// TwinCAT 3 PLC project tc_project_app
// ProgramVersion: 3.1.4024.12
// libraries:
//   Tc2_EtherCAT, * (Beckhoff Automation GmbH)
//   Tc2_MC2, * (Beckhoff Automation GmbH)
//   Tc2_Standard, * (Beckhoff Automation GmbH)
//   Tc2_SUPS, * (Beckhoff Automation GmbH)
//   Tc2_System, * (Beckhoff Automation GmbH)
//   Tc2_Utilities, * (Beckhoff Automation GmbH)
//   Tc3_MC2_AdvancedHoming, * (Beckhoff Automation GmbH)
//   Tc3_Module, * (Beckhoff Automation GmbH)
//   VisuDialogs, * (System)
// project tree:
//   DUTs/Bridge Terminal PDOs/ ST_Bridge_TSCS_OUTPUTS.TcDUT, ST_Bridge_TSCS_INPUTS.TcDUT
//   DUTs/ E_HOME_STATE.TcDUT, E_MOTION_MODE.TcDUT (not stored), E_OPERATION_MODE.TcDUT (not stored), E_OPERATION_MODE_NO.TcDUT (not stored), E_PHASE_TYPE.TcDUT (not stored), E_PWM_TYPE.TcDUT, E_PHASING_STATE_MACHINE.TcDUT (not stored), E_POSITIONING_STATE_MACHINE.TcDUT (not stored), E_VELOCITY_STATE_MACHINE.TcDUT, ST_INDRADRIVE_AXIS_COMMAND.TcDUT, ST_INDRADRIVE_AXIS_STATUS.TcDUT, ST_HW_CONTROL_ROT.TcDUT, ST_HW_CONTROL_XYZ.TcDUT, ST_HW_STATUS_DEV.TcDUT, ST_HW_STATUS_XYZ.TcDUT, ST_INDRADRIVE_IO_INPUT.TcDUT, ST_INDRADRIVE_IO_OUTPUT.TcDUT (not stored), ST_S134_MASTERCONTROLWORD.TcDUT (not stored), ST_S135_DRIVESTATUSWORD.TcDUT (not stored), ST_S144_SIGNALSTATUSWORD.TcDUT, ST_S145_SIGNALCONTROLWORD.TcDUT, ST_HW_STATUS_ROT.TcDUT, ST_STATUS_ROT.TcDUT, ST_TMS_INTERLOCKS.TcDUT, TARGET_STATE_MACHINE.TcDUT
//   / GlobalTextList.TcGTLO, PlcTask.TcTTO, PlcTaskCom.TcTTO, Visualization Manager.TcVMO (not stored)
//   GVLs/ GVL_Bridge_TSCS.TcGVL, GVL_APP.TcGVL, GVL_ErrorCodes.TcGVL, GVL_Parameters.TcGVL
//   POUs/Application_Specific/Applications/ Application_Template.TcPOU
//   POUs/Application_Specific/Axes/ Axis_Template.TcPOU, Axis_1.TcPOU, Axis_2.TcPOU, Axis_3.TcPOU
//   POUs/Bridge Terminal/FBs/ FB_Bridge_Outputs_Real.TcPOU, FB_Bridge_Inputs_Real.TcPOU, OSCAT_BYTE_OF_BIT.TcPOU, OSCAT_BYTE_TO_BITS.TcPOU, OSCAT_DW_TO_REAL.TcPOU, OSCAT_REAL_TO_DW.TcPOU
//   POUs/Bridge Terminal/ TSCS_Bridge_Inputs.TcPOU, TSCS_Bridge_Outputs.TcPOU, TSCS_Bridge_Diagnostic.TcPOU
//   POUs/Common/ChangeConfig/ FB_ReadFloatParameter.TcPOU, FB_ReadParameterInNc_v1_00.TcPOU, FB_WriteFloatParameter.TcPOU, FB_WriteParameterInNc_v1_00.TcPOU
//   POUs/Common/ErrorHandling/ DUT_ErrorState.TcDUT, FB_ErrorSystem.TcPOU (not stored), FB_GenericError.TcPOU, FB_NC_Error.TcPOU, FB_TerminalError.TcPOU, ST_ErrorEntry.TcDUT, ST_ErrorSystem.TcDUT
//   POUs/Common/GVLs_std/ GVL_back.TcGVL (not stored)
//   POUs/Common/Hardware/EtherCAT_Terminals/Analog_Inputs/ EL3174_0002.TcPOU, EL3214.TcPOU, EL3255.TcPOU, El3742.TcPOU
//   POUs/Common/Hardware/EtherCAT_Terminals/Communication/ EL6695.TcPOU
//   POUs/Common/Hardware/EtherCAT_Terminals/Digital_Inputs/ EL1008.TcPOU, EL1018.TcPOU, EL1252.TcPOU, EL1808.TcPOU, EL1809.TcPOU, EL1819.TcPOU
//   POUs/Common/Hardware/EtherCAT_Terminals/Digital_Outputs/ EL2014.TcPOU, EL2032.TcPOU, EL2252.TcPOU, EL2808.TcPOU, EL2819.TcPOU
//   POUs/Common/Hardware/EtherCAT_Terminals/Digital_Outputs/External_Types/ dutEL2521_Ctrl.TcDUT, dutEL2521_Status.TcDUT
//   POUs/Common/Hardware/EtherCAT_Terminals/Drives/ EL2522.TcPOU, EL4134.TcPOU, EL7037.TcPOU, EL7041_0052.TcPOU, EL7047.TcPOU, EL7211.TcPOU, indraDrive.TcPOU, iPOS8020.TcPOU
//   POUs/Common/Hardware/EtherCAT_Terminals/Feedback_Terminals/ EL5002.TcPOU, EL5021.TcPOU, EL5042.TcPOU, EL5101.TcPOU, EL7201.TcPOU
//   POUs/Common/Hardware/EtherCAT_Terminals/System/ EK1100.TcPOU, EK1110.TcPOU, EL9410.TcPOU, EL9505.TcPOU
//   POUs/Data Type Conversion Functions/ SCALE_REAL_TO_UDINT.TcPOU, SCALE_UDINT_TO_REAL.TcPOU
//   POUs/ MAIN_NORMAL_MOTION.TcPOU, MAIN.TcPOU
//   POUs/Target/ fbIndraDrive.TcPOU, FB_ModePhasing.TcPOU, FB_CalcVeloFromLatch.TcPOU, FB_ModeVelo.TcPOU, FB_ModePos.TcPOU, FB_ModeHome.TcPOU, FB_PID.TcPOU, FB_RampVelo.TcPOU, FB_PWM.TcPOU, FB_TargetSuperImpose.TcPOU (not stored)
//   tc_mca_std_lib_real/DUTs/ E_AxisParameters.TcTLEO (not stored), E_EncoderTypeClass.TcDUT (not stored), E_HomeSwitchTypeClass.TcDUT (not stored), E_HomingRoutines.TcTLEO (not stored), E_MotionFunctions.TcDUT (not stored), E_MotorTypeClass.TcDUT (not stored), E_RestorePosition.TcDUT (not stored), ST_AxisConfig.TcDUT (not stored), ST_AxisControl.TcDUT (not stored), ST_AxisDescription.TcDUT (not stored), ST_AxisError.TcDUT (not stored), ST_AxisInputs.TcDUT (not stored), ST_AxisPersistent.TcDUT (not stored), ST_AxisStatus.TcDUT (not stored), ST_AxisStruct.TcDUT (not stored), ST_GearAxis.TcDUT (not stored)
//   tc_mca_std_lib_real/GVLs/ GVL.TcGVL (not stored)
//   tc_mca_std_lib_real/POUs/Motion/ FB_Axis.TcPOU (not stored)
//   tc_mca_std_lib_real/POUs/Motion/Homing/ FB_Homing.TcPOU (not stored)
//   tc_mca_std_lib_real/VISUs/ languageSupport.TcTLO (not stored), MainVisu.TcVIS (not stored), visuTextLinks.TcTLO (not stored)
//   tc_pils/tc_pils_app_specific/GVLs/ GVL_PILS.TcGVL (not stored)
//   tc_pils/tc_pils_app_specific/POUs/ PILS_DEVICES.TcPOU (not stored)
//   tc_pils/tc_pils_generic/DUTs/ E_Permission.TcDUT (not stored), E_PILS_ParamControl.TcDUT (not stored), E_PILS_State.TcDUT (not stored), ST_1201.TcDUT (not stored), ST_1202.TcDUT (not stored), ST_1204.TcDUT (not stored), ST_1602.TcDUT (not stored), ST_5008.TcDUT (not stored), ST_5010.TcDUT (not stored), ST_AxisParameters.TcDUT (not stored), ST_DeviceInfo.TcDUT (not stored), ST_Indexer.TcDUT (not stored), ST_Indexer_InfoTyp0.TcDUT (not stored), ST_ParamOutput.TcDUT (not stored), U_IndexerData.TcDUT (not stored)
//   tc_pils/tc_pils_generic/POUs/ COMM.TcPOU (not stored)
//   tc_pils/tc_pils_generic/POUs/PILS_device_types/ FB_5008_Axis.TcPOU (not stored), FB_5010_Axis.TcPOU (not stored)
// real-time tasks:
//   TASK PlcTaskCom: cycle T#1ms, priority 26, ADS port 350
//   TASK PlcTask: cycle T#1ms, priority 20, ADS port 351
//   TASK Task faster: cycle T#1ms, priority 1, ADS port 352
// motion (NC):
//   TASK NC-Task 1 SAF: cycle T#2ms, priority 4, ADS port 501
//   TASK NC-Task 1 SVB: cycle T#10ms, priority 8, ADS port 511
//   AXIS Axis 1 (id 1)
//     Dynamic: AccelerationMaximum=0.15, DecelerationMaximum=0.15, Acceleration=0.02, Deceleration=0.02, Jerk=10
//     Velo: RefSearch=0.1, RefSync=0.1, SlowManual=0.01, FastManual=0.05, Maximum=0.3
//     PositionAreaControl: Range=0.2
//     TargetPosControl: Range=0.2
//     OtherSettings: AllowMotionCmdToSlave=true, PulseDistancePos=0.1, PulseDistanceNeg=0.1
//     encoder EncType=19
//       EncPara: ScaleFactorNumerator=0.340251786, ScaleFactorDenominator=51200, Inverse=true, MaxCount=#xffffffff
//     drive DrvType=16
//       DrvPara: Inverse=true, MaxCount=#xffffffff
//         Analog: VeloReferenz=0.3, VeloScale=8192, TorqueSetpointScale=10, ScaleFactorActTorque=0.1
//         TimeComp: TaskDelayCycles=1
//     controller CtrType=1
//       CtrPara: PriorControlFactor=1
//         PosDiffControl: Range=0.2, Time=0.1
//         PID: PosKp=0.1
//         Observer: BandWidth=20
//   AXIS Axis 2 (id 2)
//     Dynamic: AccelerationMaximum=0.15, DecelerationMaximum=0.15, Acceleration=0.02, Deceleration=0.02, Jerk=10
//     Velo: RefSearch=0.1, RefSync=0.1, SlowManual=0.01, FastManual=0.05, Maximum=0.3
//     PositionAreaControl: Range=0.2
//     TargetPosControl: Range=0.2
//     OtherSettings: AllowMotionCmdToSlave=true, PulseDistancePos=0.1, PulseDistanceNeg=0.1
//     encoder EncType=19
//       EncPara: ScaleFactorNumerator=0.340251786, ScaleFactorDenominator=51200, Inverse=true, MaxCount=#xffffffff
//     drive DrvType=16
//       DrvPara: Inverse=true, MaxCount=#xffffffff
//         Analog: VeloReferenz=0.3, VeloScale=8192, TorqueSetpointScale=10, ScaleFactorActTorque=0.1
//         TimeComp: TaskDelayCycles=1
//     controller CtrType=1
//       CtrPara: PriorControlFactor=1
//         PosDiffControl: Range=0.2, Time=0.1
//         PID: PosKp=0.1
//         Observer: BandWidth=20
//   AXIS Axis 3 (id 3)
//     Dynamic: AccelerationMaximum=0.03, DecelerationMaximum=0.03, Acceleration=0.01, Deceleration=0.01, Jerk=10
//     Velo: RefSearch=0.01, RefSync=0.01, SlowManual=0.01, FastManual=0.02, Maximum=0.05
//     PositionAreaControl: Range=0.01
//     TargetPosControl: Range=0.01
//     OtherSettings: AllowMotionCmdToSlave=true, PulseDistancePos=0.02, PulseDistanceNeg=0.02
//     encoder EncType=19
//       EncPara: ScaleFactorNumerator=0.011468, ScaleFactorDenominator=51200, MaxCount=#xffffffff
//     drive DrvType=16
//       DrvPara: MaxCount=#xffffffff
//         Analog: VeloReferenz=0.05, VeloScale=8192, TorqueSetpointScale=10, ScaleFactorActTorque=0.1
//         TimeComp: TaskDelayCycles=1
//     controller CtrType=1
//       CtrPara: PriorControlFactor=1
//         PosDiffControl: Range=0.01, Time=0.1
//         PID: PosKp=0.1
//         Observer: BandWidth=20
// I/O:
//   DEVICE Device 1 (EtherCAT), AmsNetId 172.30.2.35.2.1
//     Term 1 (EK1200) [EK1200-5000 EtherCAT Power supply (2A E-Bus)]
//       Term 2 (EL1809) [EL1809 16Ch. Dig. Input 24V, 3ms]
//       Term 3 (EL1809) [EL1809 16Ch. Dig. Input 24V, 3ms]
//       Term 4 (EL2819) [EL2819 16Ch. Dig. Output 24V, 0,5A, Diagnostic]
//       Term 5 (EL2819) [EL2819 16Ch. Dig. Output 24V, 0,5A, Diagnostic]
//       Term 6 (EL9505) [EL9505 Power supply terminal 5V]
//       Term 7 (EL1252-0050) [EL1252-0050 2Ch. Fast Dig. Input 5V, 1µs, DC Latch]
//       Term 8 (EL9410) [EL9410 E-Bus Power Supplier  (Diagnostics)]
//       Term 9 (EL1252) [EL1252 2Ch. Fast Dig. Input 24V, 1µs, DC Latch]
//       Term 10 (EL7201) [EL7201 1Ch. MDP742 Servo motor output stage (50V, 4A)]
//       Term 11 (EL7201) [EL7201 1Ch. MDP742 Servo motor output stage (50V, 4A)]
//       Term 12 (EL7201) [EL7201 1Ch. MDP742 Servo motor output stage (50V, 4A)]
//       Term 13 (EL3214) [EL3214 4Ch. Ana. Input PT100 (RTD)]
//       Term 18 (EL5021) [EL5021 1Ch. Sin/Cos Encoder]
//       Term 14 (EL6695) [EL6695 EtherCAT Bridge terminal (Primary)]
//       Term 15 (EL9410) [EL9410 E-Bus Power Supplier  (Diagnostics)]
//       Term 16 (EL2032) [EL2032 2Ch. Dig. Output 24V, 2A, Diagnostic]
//       Term 17 (EK1110) [EK1110 EtherCAT extension]
//     Drive 10 (IndraDrive MPB18/19) [IndraDrive MPB18/19]
//     Drive 49 (iPOS8020 BX-CAT) [iPOS8020 BX-CAT]
//     Drive 50 (iPOS8020 BX-CAT) [iPOS8020 BX-CAT]
//     Drive 51 (iPOS8020 BX-CAT) [iPOS8020 BX-CAT]
// variable links:
//   (this object) <-> Device 1 (EtherCAT)/Drive 49 (iPOS8020 BX-CAT)
//     Drive/Inputs/In/nDataIn1 <-> Transmit PDO 2 mapping parameters/Following error actual value
//     Drive/Inputs/In/nDataIn3[0] <-> Transmit PDO 1 mapping parameters/Torque (current) actual value
//     Drive/Inputs/In/nDcOutputTime <-> InfoData/DcOutputShift
//     Drive/Inputs/In/nState1 <-> Transmit PDO 1 mapping parameters/Statusword
//     Drive/Inputs/In/nState2 <-> Transmit PDO 1 mapping parameters/Statusword @bit 8
//     Drive/Inputs/In/nState4 @bit 1 <-> WcState/InputToggle
//     Drive/Inputs/In/nState4 <-> WcState/WcState
//     Drive/Outputs/Out/nCtrl1 <-> Receive PDO 1 mapping parameters/Controlword
//     Drive/Outputs/Out/nCtrl2 <-> Receive PDO 1 mapping parameters/Controlword @bit 8
//     Drive/Outputs/Out/nDataOut2 <-> Receive PDO 1 mapping parameters/Target Velocity
//     Enc/Inputs/In/nDataIn1 <-> Transmit PDO 1 mapping parameters/Position actual value
//     Enc/Inputs/In/nDataIn7 <-> Transmit PDO 3 mapping parameters/Velocity actual value
//     Enc/Inputs/In/nDcInputTime <-> InfoData/DcInputShift
//     Enc/Inputs/In/nState4 @bit 1 <-> WcState/InputToggle
//     Enc/Inputs/In/nState4 <-> WcState/WcState
//   (this object) <-> Device 1 (EtherCAT)/Drive 50 (iPOS8020 BX-CAT)
//     Drive/Inputs/In/nDataIn1 <-> Transmit PDO 2 mapping parameters/Following error actual value
//     Drive/Inputs/In/nDataIn3[0] <-> Transmit PDO 1 mapping parameters/Torque (current) actual value
//     Drive/Inputs/In/nDcOutputTime <-> InfoData/DcOutputShift
//     Drive/Inputs/In/nState1 <-> Transmit PDO 1 mapping parameters/Statusword
//     Drive/Inputs/In/nState2 <-> Transmit PDO 1 mapping parameters/Statusword @bit 8
//     Drive/Inputs/In/nState4 @bit 1 <-> WcState/InputToggle
//     Drive/Inputs/In/nState4 <-> WcState/WcState
//     Drive/Outputs/Out/nCtrl1 <-> Receive PDO 1 mapping parameters/Controlword
//     Drive/Outputs/Out/nCtrl2 <-> Receive PDO 1 mapping parameters/Controlword @bit 8
//     Drive/Outputs/Out/nDataOut2 <-> Receive PDO 1 mapping parameters/Target Velocity
//     Enc/Inputs/In/nDataIn1 <-> Transmit PDO 1 mapping parameters/Position actual value
//     Enc/Inputs/In/nDataIn7 <-> Transmit PDO 3 mapping parameters/Velocity actual value
//     Enc/Inputs/In/nDcInputTime <-> InfoData/DcInputShift
//     Enc/Inputs/In/nState4 @bit 1 <-> WcState/InputToggle
//     Enc/Inputs/In/nState4 <-> WcState/WcState
//   (this object) <-> Device 1 (EtherCAT)/Drive 51 (iPOS8020 BX-CAT)
//     Drive/Inputs/In/nDataIn1 <-> Transmit PDO 2 mapping parameters/Following error actual value
//     Drive/Inputs/In/nDataIn3[0] <-> Transmit PDO 1 mapping parameters/Torque (current) actual value
//     Drive/Inputs/In/nDcOutputTime <-> InfoData/DcOutputShift
//     Drive/Inputs/In/nState1 <-> Transmit PDO 1 mapping parameters/Statusword
//     Drive/Inputs/In/nState2 <-> Transmit PDO 1 mapping parameters/Statusword @bit 8
//     Drive/Inputs/In/nState4 @bit 1 <-> WcState/InputToggle
//     Drive/Inputs/In/nState4 <-> WcState/WcState
//     Drive/Outputs/Out/nCtrl1 <-> Receive PDO 1 mapping parameters/Controlword
//     Drive/Outputs/Out/nCtrl2 <-> Receive PDO 1 mapping parameters/Controlword @bit 8
//     Drive/Outputs/Out/nDataOut2 <-> Receive PDO 1 mapping parameters/Target Velocity
//     Enc/Inputs/In/nDataIn1 <-> Transmit PDO 1 mapping parameters/Position actual value
//     Enc/Inputs/In/nDataIn7 <-> Transmit PDO 3 mapping parameters/Velocity actual value
//     Enc/Inputs/In/nDcInputTime <-> InfoData/DcInputShift
//     Enc/Inputs/In/nState4 @bit 1 <-> WcState/InputToggle
//     Enc/Inputs/In/nState4 <-> WcState/WcState
//   tc_project_app Instance <-> Device 1 (EtherCAT)/Drive 10 (IndraDrive MPB18/19)
//     PlcTask Inputs/MAIN.dLatchedPosition <-> AT/Probe value 1 positive edge
//     PlcTask Inputs/MAIN.fbIndraDrive.stDriveStatus.nP173_MarkerPosition <-> AT/Marker position A
//     PlcTask Inputs/MAIN.fbIndraDrive.stDriveStatus.nS135_DriveStatusWord <-> AT/Drive status word
//     PlcTask Inputs/MAIN.fbIndraDrive.stDriveStatus.nS189_PositionError <-> AT/Following distance
//     PlcTask Inputs/MAIN.fbIndraDrive.stDriveStatus.nS386_ActivePositionFeedbackValue <-> AT/Active position feedback value
//     PlcTask Inputs/MAIN.fbIndraDrive.stDriveStatus.nS390_DiagnosticMessageNumber <-> AT/Diagnostic message number
//     PlcTask Inputs/MAIN.fbIndraDrive.stDriveStatus.nS40_VelocityFeedbackValue <-> AT/Velocity feedback value
//     PlcTask Inputs/MAIN.fbIndraDrive.stDriveStatus.nS51_PositionFeedbackValue <-> AT/Position feedback value 1
//     PlcTask Inputs/MAIN.fbIndraDrive.stDriveStatus.nS84_TorqueFeedback <-> AT/Torque/force feedback value
//     PlcTask Inputs/MAIN.fbIndraDrive.stDriveStatus.stS144_SignalStatusWord <-> AT/Signal status word
//     PlcTask Inputs/MAIN.fb_s19_IndraDrive.InfoData_State <-> InfoData/State
//     PlcTask Inputs/MAIN.fb_s19_IndraDrive.WcState_WcState <-> WcState/WcState
//     PlcTask Outputs/MAIN.fbIndraDrive.stDriveCommands.nS108_FeedrateOverride <-> MDT/Feedrate override
//     PlcTask Outputs/MAIN.fbIndraDrive.stDriveCommands.nS258_TargetPosition <-> MDT/Target position
//     PlcTask Outputs/MAIN.fbIndraDrive.stDriveCommands.nS259_PositioningVelocity <-> MDT/Positioning velocity
//     PlcTask Outputs/MAIN.fbIndraDrive.stDriveCommands.nS260_PositioningAcceleration <-> MDT/Ramp 1 pitch
//     PlcTask Outputs/MAIN.fbIndraDrive.stDriveCommands.nS282_PositioningCommandValue <-> MDT/Positioning command value
//     PlcTask Outputs/MAIN.fbIndraDrive.stDriveCommands.nS359_PositioningDeceleration <-> MDT/Deceleration ramp 1
//     PlcTask Outputs/MAIN.fbIndraDrive.stDriveCommands.nS40_VelocityCommandValue <-> MDT/Velocity command value
//     PlcTask Outputs/MAIN.fbIndraDrive.stDriveCommands.nS47_PositionCommandValue <-> MDT/Position command value
//     PlcTask Outputs/MAIN.fbIndraDrive.stDriveCommands.nS92_BiPolarTorqueLimit <-> MDT/Bipolar torque/force limit value
//     PlcTask Outputs/MAIN.fbIndraDrive.stDriveCommands.stS134_MasterControlWord <-> MDT/Master control word
//     PlcTask Outputs/MAIN.fbIndraDrive.stDriveCommands.stS145_SignalControlWord <-> MDT/Signal control word
//     PlcTask Outputs/MAIN.nAdditiveTorqueSetpoint <-> MDT/Additive torque/force command value
//     PlcTaskCom Outputs/MAIN.iTorqueCommandValue <-> MDT/Torque/force command value
//   tc_project_app Instance <-> Device 1 (EtherCAT)/Drive 49 (iPOS8020 BX-CAT)
//     PlcTask Inputs/MAIN.fb_s20_IPOS8020.InfoData_State <-> InfoData/State
//   tc_project_app Instance <-> Device 1 (EtherCAT)/Drive 50 (iPOS8020 BX-CAT)
//     PlcTask Inputs/MAIN.fb_s21_IPOS8020.InfoData_State <-> InfoData/State
//   tc_project_app Instance <-> Device 1 (EtherCAT)/Drive 51 (iPOS8020 BX-CAT)
//     PlcTask Inputs/MAIN.fb_s22_IPOS8020.InfoData_State <-> InfoData/State
//   tc_project_app Instance <-> Device 1 (EtherCAT)/Term 1 (EK1200)/Term 10 (EL7201)
//     PlcTask Inputs/MAIN.fb_s10_EL7201.InfoData_State <-> InfoData/State
//     PlcTask Inputs/MAIN.fb_s10_EL7201.WcState_WcState <-> WcState/WcState
//     PlcTask Inputs/MAIN.fb_s10_EL7201.fPosAct <-> FB Position/Position
//   tc_project_app Instance <-> Device 1 (EtherCAT)/Term 1 (EK1200)/Term 11 (EL7201)
//     PlcTask Inputs/MAIN.fb_s11_EL7201.InfoData_State <-> InfoData/State
//     PlcTask Inputs/MAIN.fb_s11_EL7201.WcState_WcState <-> WcState/WcState
//     PlcTask Inputs/MAIN.fb_s11_EL7201.fPosAct <-> FB Position/Position
//   tc_project_app Instance <-> Device 1 (EtherCAT)/Term 1 (EK1200)/Term 12 (EL7201)
//     PlcTask Inputs/MAIN.fb_s12_EL7201.InfoData_State <-> InfoData/State
//     PlcTask Inputs/MAIN.fb_s12_EL7201.WcState_WcState <-> WcState/WcState
//     PlcTask Inputs/MAIN.fb_s12_EL7201.fPosAct <-> FB Position/Position
//   tc_project_app Instance <-> Device 1 (EtherCAT)/Term 1 (EK1200)/Term 13 (EL3214)
//     PlcTask Inputs/MAIN.fb_s13_EL3214.InfoData_State <-> InfoData/State
//     PlcTask Inputs/MAIN.fb_s13_EL3214.WcState_WcState <-> WcState/WcState
//     PlcTask Inputs/MAIN.fb_s13_EL3214.iAI_{1..4} <-> RTD Inputs Channel {1..4}/Value  (4 links)
//     PlcTask Inputs/MAIN.fb_s13_EL3214.wCh{1..4}_Status <-> RTD Inputs Channel {1..4}/Status  (4 links)
//   tc_project_app Instance <-> Device 1 (EtherCAT)/Term 1 (EK1200)/Term 14 (EL6695)
//     PlcTask Inputs/GVL_Bridge_TSCS.INPUTS/TDU_TestSignal_RB <-> IO Inputs/TDU_WatchDog_RB
//     PlcTask Inputs/GVL_Bridge_TSCS.INPUTS/TSCS_Byte <-> IO Inputs/TSCS_Byte
//     PlcTask Inputs/GVL_Bridge_TSCS.INPUTS/TSCS_Real <-> IO Inputs/TSCS_Real
//     PlcTask Inputs/MAIN.fb_s15_EL6695.InfoData_State <-> InfoData/State
//     PlcTask Inputs/MAIN.fb_s15_EL6695.WcState_WcState <-> WcState/WcState
//     PlcTask Outputs/GVL_Bridge_TSCS.OUTPUTS/TDU_Byte <-> IO Outputs/TDU_Byte
//     PlcTask Outputs/GVL_Bridge_TSCS.OUTPUTS/TDU_Real <-> IO Outputs/TDU_Real
//     PlcTask Outputs/GVL_Bridge_TSCS.OUTPUTS/TDU_TestSignal <-> IO Outputs/TDU_WatchDog
//   tc_project_app Instance <-> Device 1 (EtherCAT)/Term 1 (EK1200)/Term 15 (EL9410)
//     PlcTask Inputs/MAIN.fb_s16_EL9410.InfoData_State <-> InfoData/State
//     PlcTask Inputs/MAIN.fb_s16_EL9410.WcState_WcState <-> WcState/WcState
//     PlcTask Inputs/MAIN.fb_s16_EL9410.bUp_Undervoltage <-> Status Up/Undervoltage
//     PlcTask Inputs/MAIN.fb_s16_EL9410.bUs_Undervoltage <-> Status Us/Undervoltage
//   tc_project_app Instance <-> Device 1 (EtherCAT)/Term 1 (EK1200)/Term 16 (EL2032)
//     PlcTask Inputs/MAIN.fb_s17_EL2032.InfoData_State <-> InfoData/State
//     PlcTask Inputs/MAIN.fb_s17_EL2032.WcState_WcState <-> WcState/WcState
//   tc_project_app Instance <-> Device 1 (EtherCAT)/Term 1 (EK1200)/Term 18 (EL5021)
//     PlcTask Inputs/MAIN.fb_s14_EL5021.InfoData_State <-> InfoData/State
//     PlcTask Inputs/MAIN.fb_s14_EL5021.WcState_WcState <-> WcState/WcState
//     PlcTaskCom Inputs/MAIN.nSecondRotEncoder <-> ENC Status/Counter value
//   tc_project_app Instance <-> Device 1 (EtherCAT)/Term 1 (EK1200)/Term 2 (EL1809)
//     PlcTask Inputs/MAIN.fb_s2_EL1809.InfoData_State <-> InfoData/State
//     PlcTask Inputs/MAIN.fb_s2_EL1809.WcState_WcState <-> WcState/WcState
//     PlcTask Inputs/MAIN.fb_s2_EL1809.bBI_{1..16} <-> Channel {1..16}/Input  (16 links)
//   tc_project_app Instance <-> Device 1 (EtherCAT)/Term 1 (EK1200)/Term 3 (EL1809)
//     PlcTask Inputs/MAIN.fb_s3_EL1809.InfoData_State <-> InfoData/State
//     PlcTask Inputs/MAIN.fb_s3_EL1809.WcState_WcState <-> WcState/WcState
//     PlcTask Inputs/MAIN.fb_s3_EL1809.bBI_{1..16} <-> Channel {1..16}/Input  (16 links)
//   tc_project_app Instance <-> Device 1 (EtherCAT)/Term 1 (EK1200)/Term 4 (EL2819)
//     PlcTask Inputs/MAIN.fb_s4_EL2819.InfoData_State <-> InfoData/State
//     PlcTask Inputs/MAIN.fb_s4_EL2819.WcState_WcState <-> WcState/WcState
//     PlcTask Inputs/MAIN.fb_s4_EL2819.bDev_CommonFault <-> DIG Inputs Device/Common Fault
//     PlcTask Inputs/MAIN.fb_s4_EL2819.bDev_MissingVoltage <-> DIG Inputs Device/Missing Voltage
//     PlcTask Inputs/MAIN.fb_s4_EL2819.bDev_Overtemperature <-> DIG Inputs Device/Overtemperature Device
//     PlcTask Inputs/MAIN.fb_s4_EL2819.bDev_UnderVoltage <-> DIG Inputs Device/Undervoltage
//     PlcTask Inputs/MAIN.fb_s4_EL2819.wCH{1..16}_Diag <-> DIG Diag Inputs/Channel {1..16}  (16 links)
//     PlcTask Outputs/MAIN.stHWControlRot.bRotOmronSensor1Feed <-> DIG Outputs/Channel 1/Output
//     PlcTask Outputs/MAIN.stHWControlRot.bRotOmronSensor2Feed <-> DIG Outputs/Channel 2/Output
//   tc_project_app Instance <-> Device 1 (EtherCAT)/Term 1 (EK1200)/Term 5 (EL2819)
//     PlcTask Inputs/MAIN.fb_s5_EL2819.InfoData_State <-> InfoData/State
//     PlcTask Inputs/MAIN.fb_s5_EL2819.WcState_WcState <-> WcState/WcState
//     PlcTask Inputs/MAIN.fb_s5_EL2819.bDev_CommonFault <-> DIG Inputs Device/Common Fault
//     PlcTask Inputs/MAIN.fb_s5_EL2819.bDev_MissingVoltage <-> DIG Inputs Device/Missing Voltage
//     PlcTask Inputs/MAIN.fb_s5_EL2819.bDev_Overtemperature <-> DIG Inputs Device/Overtemperature Device
//     PlcTask Inputs/MAIN.fb_s5_EL2819.bDev_UnderVoltage <-> DIG Inputs Device/Undervoltage
//     PlcTask Inputs/MAIN.fb_s5_EL2819.wCH{1..16}_Diag <-> DIG Diag Inputs/Channel {1..16}  (16 links)
//     PlcTask Outputs/MAIN.stHWControlX.bBrakeReleaseCmd <-> DIG Outputs/Channel 2/Output
//     PlcTask Outputs/MAIN.stHWControlX.bMinMaxFeed <-> DIG Outputs/Channel 1/Output
//     PlcTask Outputs/MAIN.stHWControlX.bMinMinMaxMaxFeed <-> DIG Outputs/Channel 3/Output
//     PlcTask Outputs/MAIN.stHWControlY.bBrakeReleaseCmd <-> DIG Outputs/Channel 6/Output
//     PlcTask Outputs/MAIN.stHWControlY.bMinMaxFeed <-> DIG Outputs/Channel 5/Output
//     PlcTask Outputs/MAIN.stHWControlY.bMinMinMaxMaxFeed <-> DIG Outputs/Channel 7/Output
//     PlcTask Outputs/MAIN.stHWControlZ.bMinMaxFeed <-> DIG Outputs/Channel 9/Output
//     PlcTask Outputs/MAIN.stHWControlZ.bMinMinMaxMaxFeed <-> DIG Outputs/Channel 10/Output
//   tc_project_app Instance <-> Device 1 (EtherCAT)/Term 1 (EK1200)/Term 6 (EL9505)
//     PlcTask Inputs/MAIN.fb_s6_EL9505.InfoData_State <-> InfoData/State
//     PlcTask Inputs/MAIN.fb_s6_EL9505.WcState_WcState <-> WcState/WcState
//     PlcTask Inputs/MAIN.fb_s6_EL9505.bUoPwr_OK <-> Status Uo/Power OK
//     PlcTask Inputs/MAIN.fb_s6_EL9505.bUo_Overload <-> Status Uo/Overload
//   tc_project_app Instance <-> Device 1 (EtherCAT)/Term 1 (EK1200)/Term 7 (EL1252-0050)
//     PlcTask Inputs/MAIN.fb_s7_EL1252.InfoData_State <-> InfoData/State
//     PlcTask Inputs/MAIN.fb_s7_EL1252.WcState_WcState <-> WcState/WcState
//     PlcTask Inputs/MAIN.fb_s7_EL1252.bBI_1 <-> Channel 1/Input
//     PlcTask Inputs/MAIN.fb_s7_EL1252.bBI_2 <-> Channel 2/Input
//   tc_project_app Instance <-> Device 1 (EtherCAT)/Term 1 (EK1200)/Term 8 (EL9410)
//     PlcTask Inputs/MAIN.fb_s8_EL9410.InfoData_State <-> InfoData/State
//     PlcTask Inputs/MAIN.fb_s8_EL9410.WcState_WcState <-> WcState/WcState
//     PlcTask Inputs/MAIN.fb_s8_EL9410.bUp_Undervoltage <-> Status Up/Undervoltage
//     PlcTask Inputs/MAIN.fb_s8_EL9410.bUs_Undervoltage <-> Status Us/Undervoltage
//   tc_project_app Instance <-> Device 1 (EtherCAT)/Term 1 (EK1200)/Term 9 (EL1252)
//     PlcTask Inputs/MAIN.fb_s9_EL1252.InfoData_State <-> InfoData/State
//     PlcTask Inputs/MAIN.fb_s9_EL1252.WcState_WcState <-> WcState/WcState
//     PlcTask Inputs/MAIN.fb_s9_EL1252.bBI_1 <-> Channel 1/Input
//     PlcTask Inputs/MAIN.fb_s9_EL1252.bBI_2 <-> Channel 2/Input
//   tc_project_app Instance <-> NC-Task 1 SAF/Axes/Axis 1
//     PlcTask Inputs/GVL.astAxes[1].Axis.NcToPlc <-> Outputs/ToPlc
//     PlcTask Outputs/GVL.astAxes[1].Axis.PlcToNc <-> Inputs/FromPlc
//   tc_project_app Instance <-> NC-Task 1 SAF/Axes/Axis 2
//     PlcTask Inputs/GVL.astAxes[2].Axis.NcToPlc <-> Outputs/ToPlc
//     PlcTask Outputs/GVL.astAxes[2].Axis.PlcToNc <-> Inputs/FromPlc
//   tc_project_app Instance <-> NC-Task 1 SAF/Axes/Axis 3
//     PlcTask Inputs/GVL.astAxes[3].Axis.NcToPlc <-> Outputs/ToPlc
//     PlcTask Outputs/GVL.astAxes[3].Axis.PlcToNc <-> Inputs/FromPlc

CONFIGURATION tc_project_app
    RESOURCE PLC ON TwinCAT3
        TASK PlcTask(INTERVAL := T#1ms, PRIORITY := 20);
        TASK PlcTaskCom(INTERVAL := T#1ms, PRIORITY := 26);
        PROGRAM MAIN WITH PlcTask : MAIN;
        PROGRAM MAIN_NORMAL_MOTION WITH PlcTask : MAIN_NORMAL_MOTION;
        PROGRAM COMM WITH PlcTaskCom : COMM;
    END_RESOURCE
END_CONFIGURATION

// ---- DUTs/Bridge Terminal PDOs/ST_Bridge_TSCS_OUTPUTS.TcDUT
TYPE ST_Bridge_TSCS_OUTPUTS :
	// 	Outputs from TDU PLC to bridge terminal (to TSCS PLC)
STRUCT
	TDU_TestSignal : UDINT;	// Diagnostic signal (for readback: This PLC -> Other PLC -> This PLC)
	TDU_Byte : ARRAY [0..3] OF BYTE; // Boolean words from TDU PLC (5x 8 Booleans)
	TDU_Real : ARRAY [0..7] OF UDINT;
END_STRUCT
END_TYPE

// ---- DUTs/Bridge Terminal PDOs/ST_Bridge_TSCS_INPUTS.TcDUT
TYPE ST_Bridge_TSCS_INPUTS :
// 	Inputs from bridge terminal (bridge with TSCS PLC)
STRUCT
	TDU_TestSignal_RB : UDINT;				// Diagnostic signal readback TDU->TSCS->TDU
	TSCS_Byte : ARRAY [0..3] OF BYTE;		// Boolean words from TSCS PLC (5x 8 Booleans)
	TSCS_Real : ARRAY [0..7] OF UDINT;
END_STRUCT
END_TYPE

// ---- DUTs/E_HOME_STATE.TcDUT
{attribute 'qualified_only'}
{attribute 'strict'}
TYPE E_HOME_STATE :
(
	IDLE      := 0,
	RAMP_UP   := 1,
	HOMING    := 2,
	RAMP_DOWN := 3
);
END_TYPE

// ---- DUTs/E_PWM_TYPE.TcDUT
{attribute 'qualified_only'}
{attribute 'strict'}
TYPE E_PWM_TYPE :
(
	NONE := 0,
	OPTIMIZED:=1,
	SIMPLE:=2
);
END_TYPE

// ---- DUTs/E_VELOCITY_STATE_MACHINE.TcDUT
{attribute 'qualified_only'}
{attribute 'strict'}
TYPE E_VELOCITY_STATE_MACHINE :
(
	POWER_OFF := 0,
	POWER_ON := 1,
	VELOCITY := 2 
);
END_TYPE

// ---- DUTs/ST_INDRADRIVE_AXIS_COMMAND.TcDUT
TYPE ST_INDRADRIVE_AXIS_COMMAND :
STRUCT
	eOperationMode				: E_OPERATION_MODE_NO	:= E_OPERATION_MODE_NO.ePrimaryOpMode;	// (S134.0-2) Defines the Operation mode to use (the different operation modes are configured in the drive) 
	bEnableAxis					: BOOL	:= FALSE; 	// FALSE (S134.13-15): Disable drive 
													// TRUE (S134.13-15): Enable drive (torque on the motor) 
	bHaltAxis					: BOOL	:= FALSE;	// FALSE (S134.13-15): Drive performs a HALT operation (Deceleration of drive while maintaining the max. acceleration (S-0-0138). Requires bEnableAxis to be TRUE) 
													// TRUE (S134.13-15): Drive is not halted
	eMotionMode					: E_MOTION_MODE		:= E_MOTION_MODE.eStop;	// Defines the type of motion that shall be performed. This is not functional in Operation Mode Drive internal interpolation! 
	//bPositioningMode			: BOOL;				// (S346.2&1 FALSE&FALSE): Activates positioning mode according to current Operation mode 
	//bJogPositive				: BOOL;				// (S346.2&1 FALSE&TRUE): Activates jogging in positive direction  
	//bJogNeagtive				: BOOL;				// (S346.2&1 TRUE&FALSE): Activates jogging in negative direction
	//bStopAxis					: BOOL;				// (S346.2&1 TRUE&TRUE): Stops the axis 
	bCommandPositionChange		: BOOL	:= FALSE;	// (S346.5) FALSE: Drive moves to current target position, before positioning to new target position (when bCommandValueAccept is toggled) 
													// (S346.5) TRUE: Immediate of target position, i.e., drive immediately acknowledges the new target position (when bCommandValueAccept is toggled) 
	fCommandPosition			: LREAL	:= 0.0;		// (S47, S258 or S282 according to OperationMode)
	fCommandVelocity			: LREAL	:= 0.0; 	// (S259): The velocity used for Positioning and Jogging
	fCommandAcceleration		: LREAL	:= 0.0;		// (S260): The acceleration used for Positioning and Jogging 
	fCommandDeceleration		: LREAL	:= 0.0;		// (S359): The deceleration used for Positioning and Jogging 
	fFeedrateOverride			: LREAL	:= 100.0; 	// (S108):  Parameter used for variable adjustment of the velocity [0..100%] 
	fTorqueLimit				: LREAL	:= 100.0;	// (S92):  Parameter used for limiting the torque [0..drive/motor limit%] 
	bPositionCommandValue		: BOOL	:= FALSE;	// (S346.3): FALSE: Command position is absolute 
													// (S346.3): TRUE: Command position is relative
	bCommandValueAccept			: BOOL	:= FALSE; 	// (S346.0) Toggle bit (FALSE->TRUE or TRUE->FALSE) to start a positioning command in Operation mode "Drive controlled Positioning"
	bCmd_ErrorReset				: BOOL	:= FALSE;	// (S99): Reset the error of the drive 
	bCmd_SetAbsolutePosition	: BOOL	:= FALSE;	// (P12, C0300): Sets the Absolute position of the drive according to drive configuration 
	bCmd_DriveControlledHoming	: BOOL	:= FALSE;	// (S148, C0600): Starts the homing procedure configured in the drive. NOTE that this does not set the absolute position 
	bCmd_DisableLimits			: BOOL	:= FALSE;	// (bS159, C1300): Disables Monitoring of Position error, Position command error, Velocity error and Acceleration limit
	bCmd_ActivateParameterMode	: BOOL	:= FALSE;	// (S420, C0400): TRUE: Brings the drive to parameter mode 
	bCmd_ExitParameterMode		: BOOL	:= FALSE;	// (S422, C0200): TRUE: Brings the drive from parameter mode 
	bCmd_RunVirtualMater		: BOOL	:= FALSE;	// Jog command to the virtual Master
	bCmd_NCHomeEnable           : BOOL  := FALSE;   // Home from master NC enable (to be able to latch ref marks)
    bCmd_GetMarkerPosition      : BOOL  := FALSE;   // Start command C1400 Get Marker Position
	fVelocityCommandValue		: LREAL	:= 0.0; 	// (S40): The velocity used for Positioning and Jogging
END_STRUCT
END_TYPE

// ---- DUTs/ST_INDRADRIVE_AXIS_STATUS.TcDUT
TYPE ST_INDRADRIVE_AXIS_STATUS :
STRUCT

	bDriveInParameterMode		: BOOL;		// FALSE (S424): Drive is in Operating mode
											// TRUE (S424): The drive is in parameter mode (parameterization level 1 is active)
	eActualOperationModeNo		: E_OPERATION_MODE_NO	:= E_OPERATION_MODE_NO.ePrimaryOpMode;	// (S134.0-2) Defines the Operation mode to use (the different operation modes are configured in the drive) 
	bDCBusPresent				: BOOL;		// FALSE: DC-bus is not present (drive status bb)
											// TRUE (S135.1&0 TRUE&FALSE): DC-bus present (drive state Ab)
	bAxisEnabled				: BOOL; 	// TRUE (S135.1&0 TRUE&TRUE): Axis is operational with torque (drive state AF)
	bAxisHomedStatus			: BOOL; 	// TRUE (S403.0): Axis absolute position is established 
	bAxisStandStillStatus		: BOOL;		// TRUE (S331): Axis is standing still (velocity below configured threshold) 
	bAxisInTargetPosition		: BOOL;		// TRUE (S437.2): Axis command position is reached
	bAxisConstantVelocityStatus	: BOOL;		// TRUE (S437.4): Axis in constant velocity
	bAxisAccelerationStatus		: BOOL;		// TRUE (S437.5): Axis in acceleration
	bAxisDecelerationStatus		: BOOL;		// TRUE (S437.6): Axis in deceleration
	bAxisJogStatus				: BOOL;		// TRUE (S437.12): Axis in jog mode
	fActualPosition				: LREAL;	// The actual position of the axis
	fActualVelocity				: LREAL;	// The actual velocity of the axis
	fActualTorque				: LREAL;	// The actual torque of the axis
	fPositionError				: LREAL;	// The position error of the axis, i.e. the deviation between the Axis Set position and Actual position
	fMarkerPosition             : LREAL;
    bCommandChange				: BOOL;		// (S135.5): Bit that toggle every time a new command has been recognised by the drive 
	bCommandValueProcessing		: BOOL;		// FALSE (S115.3): Drive ignores (external) command value input (S47, S258, S282 etc) 
											// TRUE (S115.3): Drive follows (external) command value input (S47, S258, S282 etc) 
	bSTOActiveCh1   			: BOOL;     // FALSE: STO OK (motor can run)
	                                        // TRUE:  STO is active
	bSTOActiveCh2   			: BOOL;     // FALSE: STO OK (motor can run)
	                                        // TRUE:  STO is active
    bLimitsDisabled				: BOOL;		// TRUE (S159-C1300): 	Monitoring of Position error, Position command error, Velocity error and Acceleration limit is disabled
											// FALSE (S159-C1300): 	Monitoring of Position error, Position command error, Velocity error and Acceleration limit is enabled 
	bDiagMessage				: BOOL;		// TRUE (S135.11): There is a Diagnostic message on the drive 
	bWarning					: BOOL;		// TRUE (S135.12): There is a warning present on the drive 
	bError 						: BOOL;		// TRUE (S135.13): There is an error present on the drive 
	bCmd_GetMarkerPositionDone  : BOOL;     // C1400 command Get Marker Position done
	nDiagMessage				: DWORD;	// (S390) Displays the actual diagnostic message on the drive 
END_STRUCT
END_TYPE

// ---- DUTs/ST_HW_CONTROL_ROT.TcDUT

TYPE ST_HW_CONTROL_ROT :
STRUCT
	bRotOmronSensor1Feed AT %Q* :BOOL;  // s4: ch1: Feed omron sensor 1
	bRotOmronSensor2Feed AT %Q* :BOOL;  // s4: ch2: Feed omron sensor 2
	bManualInterlockOverride: BOOL:=FALSE;
	bExecute          : BOOL:=FALSE;
	bEnable           : BOOL:=FALSE;
	bReset            : BOOL:=FALSE;
	fVelSet           : LREAL:=0;
	fPosSet           : LREAL:=0;
	eTargetStateCmd   : TARGET_STATE_MACHINE:=TARGET_STATE_MACHINE.NONE;
	ePhaseCntrlAlg    : E_PHASE_TYPE:=E_PHASE_TYPE.PID;
	ePhasePwmType     : E_PWM_TYPE:=E_PWM_TYPE.NONE;
	fPhaseOffsetMM    : LREAL:=0;
	bAllowMotionGUI   : BOOL:=FALSE;       // Allow motion from GUI
	//brake: Only in test rig
	//bBrakeLockOnCmd   : BOOL:=FALSE;
	//bFreeWheelOnOnCmd : BOOL:=TRUE;
	//fBrakeSpNm        : LREAL:=0;
END_STRUCT
END_TYPE

// ---- DUTs/ST_HW_CONTROL_XYZ.TcDUT

TYPE ST_HW_CONTROL_XYZ :
STRUCT
	bMinMaxFeed  AT %Q* :BOOL;         // s5: ch1: kf05: w02.bg01 w02.bg02 stepper x limit switch max, limit min
	bBrakeReleaseCmd  AT %Q* :BOOL;    // s5: ch2: kf05: w02.ql1: stepper x brake ONLY x and Y
	bMinMinMaxMaxFeed  AT %Q* :BOOL;   // s5: ch3: kf05: w02.bg03 w02.bg04 stepper x limit switch max max, limit min min
    bManualInterlockOverride: BOOL:=FALSE;
	bAllowMotionGUI:BOOL:=FALSE;       // Allow motion from GUI
	bExecuteAbsPos:BOOL:=FALSE;
	bExecuteConstVelo:BOOL:=FALSE;
	bExecuteHome:BOOL:=FALSE;
	bExecuteStop:BOOL:=FALSE;
	bEnable:BOOL:=FALSE;
	bExecuteReset:BOOL:=FALSE;
	bJogDirFwd:BOOL:=1;   // 1=fwd, 0=bwd
END_STRUCT
END_TYPE

// ---- DUTs/ST_HW_STATUS_DEV.TcDUT
// HW status for control cabinet alarms and rotation drive
TYPE ST_HW_STATUS_DEV :
STRUCT	
	bEStopOK:BOOL;                       // s2: ch1: emergency stop ok                 Verify: OK   
	bRF02_MainDriveThermalFilterOK:BOOL; // s2: ch2: rf01 termal braking filter OK..   Verify: Q to Markus: Maybe this should be rf02?
	bTA01_TA02_24VSupplyOK:BOOL;         // s2: ch3: ta01 and ta02 24V power supply OK Verify: OK  
	bFC11_Fuse24VOK:BOOL;                // s2: ch4: fc11 24V fuse OK                   Verify: OK
	bFA01_FA02_OvervoltageOK:BOOL;       // s2: ch5: fa01 and fa02 overvoltage protection OK
	bFC01_FuseMainRotationOK:BOOL;       // s2: ch6: fc01 fuse target wheel motor OK
	bFC06_FC07_FuseICSOutletsOK:BOOL;    // s2: ch7: fc06 and fc07 ICS outlets fuse OK
	bFC51_FC52_FC53_FuseUPSOK:BOOL;      // s2: ch8: fc51, fc52 and fc53 UPS fuses OK (something wrong)
	
	// Bridge terminal EL6695
	bBeamOff:BOOL; 
	
END_STRUCT
END_TYPE

// ---- DUTs/ST_HW_STATUS_XYZ.TcDUT
// HW status for XYZ axis
TYPE ST_HW_STATUS_XYZ :
STRUCT
	bEStopOK:BOOL;
	fStepperTemp: LREAL;
	bLimitMax:BOOL;
	bLimitMin:BOOL;
	bLimitMaxMax:BOOL;
	bLimitMinMin:BOOL;
	bSumBwdILOK:BOOL:=FALSE;   
	bSumFwdILOK:BOOL:=FALSE;  
	bManualInterlockOverride:BOOL;
	bHwStatusOK:BOOL;  // Status of hardware (IPOS, EL7201, EL3214, fuses..)
	bGeneralILOK:BOOL:=FALSE;  // All on direction related summary interlocks
	bGeneralAndOverrideILOK:BOOL:=FALSE;
	bBusy:BOOL:=FALSE;
	bEnabled:BOOL:=FALSE;
	bHomed:BOOL:=FALSE;
	bHomingCmdActive:BOOL:=FALSE;
	
	// Position Outside range alarms
	bHiAlm:BOOL:=FALSE;
	bHiHiAlm:BOOL:=FALSE;
	bLoAlm:BOOL:=FALSE;
	bLoLoAlm:BOOL:=FALSE;
	
	//Only X and Y
	bBrakeReleased: BOOL;
	
	//Only for Z
    bLimitMinPark:BOOL;
	bLimitMinMinPark:BOOL;	
	bParkingRangeEnabled:BOOL;
END_STRUCT
END_TYPE

// ---- DUTs/ST_INDRADRIVE_IO_INPUT.TcDUT
TYPE ST_INDRADRIVE_IO_INPUT :	// Contains the data that is read from the drive
STRUCT
	nS135_DriveStatusWord				AT %I*	: ST_S135_DRIVESTATUSWORD; 
	nS51_PositionFeedbackValue			AT %I*	: DINT; 
	nS386_ActivePositionFeedbackValue	AT %I*	: DINT; 
	nS40_VelocityFeedbackValue			AT %I*	: DINT; 
	nS390_DiagnosticMessageNumber		AT %I*	: DWORD; 
	stS144_SignalStatusWord				AT %I*	: ST_S144_SIGNALSTATUSWORD;
	nS84_TorqueFeedback					AT %I*	: INT;
	nS189_PositionError					AT %I*	: DINT;
	nP173_MarkerPosition                AT %I*  : DINT;
END_STRUCT
END_TYPE

// ---- DUTs/ST_S144_SIGNALSTATUSWORD.TcDUT
TYPE ST_S144_SIGNALSTATUSWORD :
STRUCT
	bS424_DriveMode						: BIT; 	// FALSE: Operating mode
												// TRUE: Parameter mode
	{attribute 'hide'}
	bS144_1_NotDefined					: BIT;
	bS403_0_AxisHomedStatus				: BIT; 	// FALSE: Axis is NOT homed 
												// TRUE: Axis is homed
	bS331_StandStillStatus				: BIT; 	// FALSE: Axis is moving
												// TRUE: Axis is standing still 
	bS437_2_CommandPositionReached		: BIT; 	// FALSE: Axis is NOT not within command position
												// TRUE: Axis has reached command position
	{attribute 'hide'}
	bS144_5_NotDefined					: BIT;
	{attribute 'hide'}
	bS144_6_NotDefined					: BIT;
	bP115_3_StatusOfCmdValueProcessing	: BIT; 	// FALSE: Drive ignores external command value input 
												// TRUE: Drive follows external command value input
	
	bP106_1_STO_ch1 					: BIT;  // FALSE: STO OK (motor can run)
	                                            // TRUE:  STO is active
	bP106_2_STO_ch2 					: BIT;  // FALSE: STO OK (motor can run)
	                                            // TRUE:  STO is active
	bS419_0_PositioningCmdAck			: BIT; 	// Toggled as soon as the new Position Command value is accepted and effective
	bS437_4_ConstantVelocity			: BIT; 	// TRUE: Axis in constant velocity
	bS437_5_Acceleration				: BIT; 	// TRUE: Axis in acceleration
	bS437_6_Deceleration				: BIT; 	// TRUE: Axis in deceleration
	bS437_12_JogMode					: BIT; 	// TRUE: Axis in Axis in jog mode
	//{attribute 'hide'}
	//bS144_15_NotDefined					: BIT;	
	bP14_0_C1400_GetMarkerPositionDone  : BIT   := FALSE;
END_STRUCT
END_TYPE

// ---- DUTs/ST_S145_SIGNALCONTROLWORD.TcDUT
TYPE ST_S145_SIGNALCONTROLWORD :
STRUCT
	bS346_0_PosCtrlWord_CmdValueAccept		: BIT	:= FALSE; 	// Toggle to execute Slave Axis command
	bP12_C300_SetAbsolutePosition			: BIT	:= FALSE;	// Sets the Absolute position (defined in S52) of the drive
	bS148_C600_DriveControlledHoming		: BIT	:= FALSE; 	// Initiates the homing procedure defined in the drive
	bS346_3_PosCtrlWord_Abs_Rel				: BIT	:= FALSE;	// FALSE: Absolute 
																// TRUE: Relative									
	bS346_5_PosCtrlWord_ImmBlockChange		: BIT	:= FALSE;	// FALSE: Drive moves to current target position, before positioning at new target position
																// TRUE: Immediate block change, i.e., drive immediately moves to new target position
	bS99_DriveErrorReset					: BIT	:= FALSE;	
	bS346_1_PosCtrlWord_PosActivation		: BIT	:= FALSE;	// (bS346_2 | bS346_1) 00:	Positioning active, started by toggling of bit 0
																// (bS346_2 | bS346_1) 01: 	Infinite travel in positive direction (jog+) (Positioning will be aborted)
																// (bS346_2 | bS346_1) 10: 	Infinite travel in negative direction (jog-) (Positioning will be aborted)
																// (bS346_2 | bS346_1) 11: 	Stopping the axis (positioning stop) (Positioning will be aborted)
	bS346_2_PosCtrlWord_PosActivation		: BIT	:= FALSE;	// (bS346_2 | bS346_1) 00:	Positioning active, started by toggling of bit 0
																// (bS346_2 | bS346_1) 01: 	Infinite travel in positive direction (jog+) (Positioning will be aborted)
																// (bS346_2 | bS346_1) 10: 	Infinite travel in negative direction (jog-) (Positioning will be aborted)
																// (bS346_2 | bS346_1) 11: 	Stopping the axis (positioning stop) (Positioning will be aborted)
	                 	
	bS159_C1300_Disable_Monitoring			: BIT	:= FALSE;	// TRUE: 	Monitoring of Position error, Position command error, Velocity error and Acceleration limit is disabled
																// FALSE: 	Monitoring of Position error, Position command error, Velocity error and Acceleration limit is enabled 
	                  	
	bS405_0_Probe1_Enabled					: BIT	:= TRUE;
	bS420_C0400_Activate_ParameterMode		: BIT	:= FALSE;	// Brings the drive into parameter mode
	bS422_C0200_Exit_ParameterMode			: BIT	:= FALSE;	// Brings the drive into parameter mode
	bP760_VM_PosCtrlWord_CmdValueAccept		: BIT	:= FALSE;	// Toggle to execute Virtual Master command
	bP760_VM_PosCtrlWord_1_PosActivation	: BIT	:= FALSE;	// (bP760_2 | bP760_1) 00:	Positioning active, started by toggling of bit 0
																// (bP760_2 | bP760_1) 01: 	Infinite travel in positive direction (jog+) (Positioning will be aborted)
																// (bP760_2 | bP760_1) 10: 	Infinite travel in negative direction (jog-) (Positioning will be aborted)
																// (bP760_2 | bP760_1) 11: 	Stopping the axis (positioning stop) (Positioning will be aborted)
	//bP760_VM_PosCtrlWord_2_PosActivation	: BIT	:= FALSE;	// (bP760_2 | bP760_1) 00:	Positioning active, started by toggling of bit 0
																// (bP760_2 | bP760_1) 01: 	Infinite travel in positive direction (jog+) (Positioning will be aborted), started by toggling of bit 0
																// (bP760_2 | bP760_1) 10: 	Infinite travel in negative direction (jog-) (Positioning will be aborted), started by toggling of bit 0
																// (bP760_2 | bP760_1) 11: 	Stopping the axis (positioning stop) (Positioning will be aborted)
	//{attribute 'hide'}
	//bS145_15_NotDefined						: BIT	:= FALSE;
	
	//Bit 15
	bS407_0_HomingEnbale                    : BIT   := FALSE;
	//Bit 16
	bP14_0_C1400_GetMarkerPosition          : BIT   := FALSE;  
END_STRUCT
END_TYPE

// ---- DUTs/ST_HW_STATUS_ROT.TcDUT
TYPE ST_HW_STATUS_ROT :
STRUCT
	bError:BOOL:=FALSE;
	nErrorId:UDINT:=0;
	bEnabled:BOOL:=FALSE;
	eTargetState: TARGET_STATE_MACHINE;
    sErrorStr:STRING:='NO ERROR';
	fActTorque:LREAL:=0;
	fActPos:LREAL:=0;
	fActVel:LREAL:=0;	
	fActTemp:LREAL:=0;
	fSetVelRaw:LREAL;
	fBrakeActTemp1:LREAL;
	fBrakeActTemp2:LREAL;
	fPhaseOffsetActDeg:LREAL;
	bEStopOK:BOOL;                       // s2: ch1: emergency stop ok                 Verify: OK   
	bMainDriveThermalFilterOK:BOOL; // s2: ch2: rf01 termal braking filter OK..   Verify: Q to Markus: Maybe this should be rf02?
	bFuseMainRotationOK:BOOL;       // s2: ch6: fc01 fuse target wheel motor OK
	fRotTemp:LREAL;                 // s13: ch4: kf12 Target Main motor Temperature (KTY) (in deg*10)
	bSumILOK:BOOL:=FALSE;
	bHwStatusOK:BOOL:=FALSE;
	bManualInterlockOverride:BOOL:=FALSE;
	bGeneralILOK:BOOL:=FALSE;  // All on direction related summary interlocks
	bHomed:BOOL:=FALSE;
END_STRUCT
END_TYPE

// ---- DUTs/ST_STATUS_ROT.TcDUT
TYPE ST_STATUS_ROT :
STRUCT
		bPhaseOK:BOOL:=FALSE;
END_STRUCT
END_TYPE

// ---- DUTs/ST_TMS_INTERLOCKS.TcDUT
TYPE ST_TMS_INTERLOCKS :
STRUCT
	TSM_RotIL_XY_OK:BOOL:=FALSE;
	TSM_RotIL_Z_OK:BOOL:=FALSE;
	TSM_RotIL_BearTmp_OK:BOOL:=FALSE;
	TSM_RotIL_Vibr_OK:BOOL:=FALSE;	
END_STRUCT
END_TYPE

// ---- DUTs/TARGET_STATE_MACHINE.TcDUT
{attribute 'qualified_only'}
{attribute 'strict'}
TYPE TARGET_STATE_MACHINE :
(
	NONE              := 0,
	CONSTANT_VELOCITY := 2,
	POSITIONING       := 3,
	PHASING           := 4,
	HOMING            := 5,
	TORQUE            := 6
);
END_TYPE

// ---- POUs/Common/ErrorHandling/DUT_ErrorState.TcDUT
{attribute 'qualified_only'}
{attribute 'strict'}
TYPE DUT_ErrorState :
(
    None,
    Active,
    Inactive,
    Acknowledged
);
END_TYPE

// ---- POUs/Common/ErrorHandling/ST_ErrorEntry.TcDUT
TYPE ST_ErrorEntry :
STRUCT
    ErrorNum    : ULINT := 0;               //ID of the Error entry
    ErrorState  : DUT_ErrorState;           //State of the error

    //Error related
    iTerminalID     : INT;                  //ID of the terminal
    sDateTimeOn     : STRING(24);           //Date and time when the error occured
    sDateTimeOff    : STRING(24);           //Date and time when the error disapeared
    sErrorMessage   : STRING (128);         //Description of the event

    ErrorPriority   : INT;                  //Priority of the error
END_STRUCT
END_TYPE

// ---- POUs/Common/ErrorHandling/ST_ErrorSystem.TcDUT
TYPE ST_ErrorSystem :
STRUCT
    //Array of error data. Size = cSizeOfErrorData in the GVL
    aErrorData      : ARRAY [0..cSizeOfErrorData - 1] OF ST_ErrorEntry;     //Error Entry List
    nNextErrorNum   : ULINT := 1;                   //ErrorID for the next error entry
    nNoError        : UINT;                         //Number of errors in the list
    nNoActive       : UINT;                         //Number of Active errors
    nNoInactive     : UINT;                         //Number on Inactive errors
    nNoFree         : UINT;                         //Number of free entries in the list
    nNoOverflow     : INT := 0;                     //Number of overflows. How many error entries have been lost due to the size of the array
END_STRUCT
END_TYPE

// ---- POUs/Common/Hardware/EtherCAT_Terminals/Digital_Outputs/External_Types/dutEL2521_Ctrl.TcDUT
TYPE dutEL2521_Ctrl :
STRUCT
    ///The control word (CW) is located in the output process image, and is transmitted from the controller to the terminal.
    ///CW.0 FREQ_SEL 0bin / 1bin  Rapid change of the base frequency (only if the ramp function is inactive):
    ///0bin = Base frequency 1 (object 8001:02)
    ///1bin = Base frequency 2 (object 8001:03)
    FREQ_SEL: BOOL;
    ///CW.1 RAMP_DIS 1bin Operation of the ramp function is cancelled, in spite of object 8000:06 being active; if travel distance control is active, it is interrupted by this bit
    RAMP_DIS: BOOL;
    ///CW.2 GO_COUNTER 1bin  If travel distance control is active (object 8000:0A), then a pre-set counter value is approached when the bit is set
    GO_COUNTER: BOOL;
    ///CW.5 CNT_CLR 1bin The contents of the counter is cleared or set (object 8000:0B) by this bit.
    ///Any overflow or underflow bits that might be set are also cleared by this bit.
    ///The process can be edge triggered or level triggered (object 8000:05).
    CNT_CLR: BOOL;
END_STRUCT
END_TYPE

// ---- POUs/Common/Hardware/EtherCAT_Terminals/Digital_Outputs/External_Types/dutEL2521_Status.TcDUT
TYPE dutEL2521_Status :
STRUCT
    ///The status word (SW) is located in the input process image, and is transmitted from the terminal to the controller.
    ///SW.0 SEL_ACK/END_COUNTER 1bin  Confirms the change of base frequency. At activated travel distance control: target counter value reached
    SEL_ACK: BOOL;
    ///SW.1 RAMP_ACTIVE 1bin Ramp is currently being followed
    RAMP_ACTIVE: BOOL;
    ///SW.2 UNDERFLOW 1bin This bit is set if the 16-bit counter underflows (0 -> 65535). It is reset when the counter drops below two thirds of its measuring range (43690 -> 43689) or immediately an overflow occurs.
    UNDERFLOW: BOOL;
    ///SW.3 OVERFLOW 1bin This bit is set if the 16-bit counter overflows (65535 -> 0). It is reset when the counter exceeds one third of its measuring range (21845 -> 21846) or immediately an underflow occurs
    OVERFLOW: BOOL;
    ///SW.4 INPUT_T 1bin Status of INPUT_T
    INPUT_T: BOOL;
    ///SW.5 INPUT_Z 1bin Status of INPUT_Z
    INPUT_Z: BOOL;
    ///SW.6 ERROR 1bin General error bit, included with overflow/underflow
    ERROR: BOOL;
END_STRUCT
END_TYPE

// ---- GVLs/GVL_Bridge_TSCS.TcGVL
{attribute 'qualified_only'}
VAR_GLOBAL
	INPUTS  AT %I* : ST_Bridge_TSCS_INPUTS;		// Inputs
	OUTPUTS AT %Q* : ST_Bridge_TSCS_OUTPUTS;	// Outputs
END_VAR

// ---- GVLs/GVL_APP.TcGVL
{attribute 'qualified_only'}
VAR_GLOBAL CONSTANT
	nAXIS_NUM:INT:=3;
END_VAR

// ---- GVLs/GVL_ErrorCodes.TcGVL
{attribute 'qualified_only'}
VAR_GLOBAL
  // ************************General****************************	
  nErrorCodeOKId              : UDINT  := 0;
  nErrorCodeOKStr             : STRING := 'NO ERROR';
  // To high velocity 
  nErrorVelToHigh             : UDINT  := 100;
  sErrorVelToHigh             : STRING := 'MAIN: VELOCITY TO HIGH';
  //Invalid state choosen
  nErrorInvalidState          : UDINT  := 101;
  sErrorInvalidState          : STRING := 'MAIN: Invalid state';
  
  // ************************FB_ModePhase()****************************	
  // No new latched position value have been identified for the last 71 ms (no signal from timing system?)
  nErrorNoLatchId             : UDINT  := 1000;
  sErrorNoLatchStr            : STRING := 'PHASE: NO LATCH FROM DRIVE';
	
  // ************************FB_ModeHome()*****************************
  // The encoder index pulse seems to be lost (a latch have not been identified for the last rev)
  nErrorEncoderLatchLost      : UDINT  := 2000;
  sErrorEncoderLatchLost      : STRING := 'HOME: ENCODER INDEX PULSE LATCH LOST';
  // Deviation found in the latched position values (on index pulse)
  // Could be that encoder pulses are lost or that several index latches occurs per rev.
  nErrorEncoderLatchMissMatch : UDINT  := 2001;
  sErrorEncoderLatchMissMatch : STRING := 'HOME: ENCODER INDEX PULSES POSITION MISSMATCH';
  
  // ************************Indrdradrive*****************************
  nErrorIndraNotReady    : UDINT  := 3000;
  sErrorIndraNotReady    : STRING := 'INDRA: Not ready. Check status of drive (DC-BUS, STO, Tempereature...)';
  nErrorIndraTempToHigh  : UDINT  := 3001;
  sErrorIndraTempToHigh  : STRING := 'INDRA: Motor temperature to high.';
  // Drive not enable
  nErrorNotEnabled       : UDINT  := 3002;
  sErrorNotEnabled       : STRING := 'INDRA: Drive not enabled';
  // Connection lost or re param, need to be re homed
  nErrorNeedHoming       : UDINT  := 3003;
  sErrorNeedHoming       : STRING := 'INDRA: Drive need homing (re param or lost conenction)';
  //Indradrive overheat prewarning
  nErrorIndraOverHeatPrewarning       : UDINT  := 3004;
  sErrorIndraOverHeatPrewarning       : STRING := 'INDRA: Overheat prewarning';
  //Indradrive warning
  nErrorIndraWarning       : UDINT  := 3005;
  sErrorIndraWarning       : STRING := 'INDRA: Warning';
  
END_VAR

// ---- GVLs/GVL_Parameters.TcGVL
{attribute 'qualified_only'}
VAR_GLOBAL
  fSpeedToleranceRpm: LREAL := 0.05;
END_VAR

VAR_GLOBAL CONSTANT
  // Sectors of wheel	
  nSectors                             : LREAL := 36;
  // Pulse frequency
  nPulseFreqHz                         : LREAL := 14;
  // Nominal velocity of wheel
  fNominalSpeedRpm                     : LREAL := GVL_Parameters.nPulseFreqHz/GVL_Parameters.nSectors*60;
  // Velocity offset, to compensate for differnce in drive and timing system
  fNominalSpeedAdjust                  : LREAL:=0.001;//-0.0002;  //Timing system vs drive clock tuning. Automize later!
  // Speed for last revs needs to be below this value before start to phase 
  fPhaseSpeedTol                       : LREAL := 0.05;
  // Velocity setpoint for homing 
  fHomeSpeedRpm: LREAL := 5;
  // Maximum allowed speed
  fMaximumSPeedRpm: LREAL := 28;
  fMaximumSPeedSPRpm: LREAL := 25;
  nMaxMotorTemperature: INT:= 90;
  nMaxBrakeTemperature: INT:= 100;
  fWheelDiameter:LREAL:=2500;
  fAccDefaultVel:LREAL:=0.039;  //RPM/S^2 (0.039 => tn min to 23.3) 
  fAccDefaultPos:LREAL:=0.001;  //RPM/S^2 (0.039 => tn min to 23.3) 
  nPhaseErrorFilterSize:INT:=36;  //Two revs
  nVeloInRangeCount:INT:=100;
  nSuperPosMaxCyclesToOutput:INT:=100;
  fSuperPosDutyCycle:LREAL:=2.0/3.0;
  nTaskSampleTime:INT:=1;
  nPhasePIDReducedSampleRateFactor:INT:=1;   //run pid every time new pulse
  nRefMarkArraySize:UDINT:=10;
  fCheckTimingPulseMinVel: LREAL:=2.0;
  fMaxPhaseOffsetMM : LREAL:=100;
  fMinPhaseOffsetMM : LREAL:=-100;
  fMinVelSetpointAbsRpm : LREAL:=2;
  fNominalFFTourqueAbs:LREAL:=62;  //62%
  fStartupFFTourqueAbs:LREAL:=150;  //62%
  fMaxRotationBipolarTorque: LREAL :=200.0;  //Max indra drive torque
  
  // Use this var to calibrate offset from alignment.
  fRotPosOffsetDeg : LREAL :=195;  // Offset between encoder 0 and centre of sector 1 (centre of home sensor hole in direction X)
  
  // ESS-0127013 requirements
  //   FR31 Starnge to require a setting like this for commisioning.. but OK.
  bTargetRotorInstalled: BOOL:=TRUE;
  
  // Need to set resonable values here
  fXRangeH1:LREAL:=4;    // High
  fXRangeH2:LREAL:=5;  // High high
  fXRangeL1:LREAL:=-4;   // Low
  fXRangeL2:LREAL:=-5; // Low low
  fYRangeH1:LREAL:=4;
  fYRangeH2:LREAL:=5;
  fYRangeL1:LREAL:=-4;
  fYRangeL2:LREAL:=-5;
  fZRangeH1:LREAL:=4;
  fZRangeH2:LREAL:=5;
  fZRangeL1:LREAL:=0;
  fZRangeL2:LREAL:=-1;
  fZRangeParkL1:LREAL:=-1.0;
  fZRangeParkL2:LREAL:=-1.1;
  
  fXStepperTargetVelo:LREAL:=0.2;
  fXStepperTargetAcc:LREAL:=0.1;
  
  fYStepperTargetVelo:LREAL:=0.2;
  fYStepperTargetAcc:LREAL:=0.1;
  
  fZStepperTargetVelo:LREAL:=0.03;
  fZStepperTargetAcc:LREAL:=0.01;
  
  fStepperTempH2:LREAL:=120;  // Deg C
  
  fXHomePosition:LREAL:=21.0;
  fYHomePosition:LREAL:=21.0;
  fZHomePosition:LREAL:=7.5;
  
  fXHomeVelOffCam:LREAL:=0.02;
  fYHomeVelOffCam:LREAL:=0.02;
  fZHomeVelOffCam:LREAL:=0.01;
  
  fXHomeVelToCam:LREAL:=0.05;
  fYHomeVelToCam:LREAL:=0.05;
  fZHomeVelToCam:LREAL:=0.03;
  
  // Phase OK calcs
  timePhaseStabilizationTime:TIME:=T#60S;
  timePhaseGreaterThanH1Time:TIME:=T#10S;
  fPhaseStabilityVelocityLowLinit:LREAL:=20.0;
  fNominalPhaseErrorLimitMM:LREAL:=2.0;
  fH1PhaseErrorLimitMM:LREAL:=5.0;
  fH2PhaseErrorLimitMM:LREAL:=10.0;
  
END_VAR

// ---- POUs/MAIN.TcPOU
PROGRAM MAIN
VAR
	
	hmiAxisSelection: INT := 1; //Not possible to use local hmi variables for array indexes
    afbAxes: ARRAY [1..GVL_APP.nAXIS_NUM] OF FB_Axis;
	stAmsNetId	AT %I*	              : AMSNETID;
	nPort	AT %I*                    : WORD;
	nMasterAxisPosition AT %I*        : DINT;
	nMainDriveMarkPosition AT %I*     : DINT;
	nAdditiveTorqueSetpoint    AT %Q* : INT;   // Unit 0.1%  (10=1%)
	dLatchedPosition AT %I*           : DINT;
	inputDigSens1 AT %I*              : BOOL;
	inputDigSens2 AT %I*              : BOOL;
	nSecondRotEncoder AT %I*           :UDINT:=0;
	fbModePhase                       : FB_ModePhasing;	 // Phasing Mode
	fbRampVelo                        : FB_RampVelo;
	fbModeVelo                        : FB_ModeVelo;     // Velocity Mode
	fbModePos                         : FB_ModePos;      // Positioning Mode
	fbModeHome                        : FB_ModeHome;     // Homing Mode
	fbCalcVeloLatch                   : FB_CalcVeloFromLatch;
	fbIndraDrive                      : fbIndraDrive;    // Control of drive
	stCommands                        : ST_INDRADRIVE_AXIS_COMMAND; // Control to drive
	stStatus                          : ST_INDRADRIVE_AXIS_STATUS;  // Status from drive
	eTargetStateOld                   : TARGET_STATE_MACHINE;
	addStartupTorqueTrigger           : BOOL:=FALSE;
	iTorqueCommandValue  AT %Q*       : INT := 0;
	bApplyTorqueFF                    : BOOL := FALSE;
	nTest: INT;
	bRotImportantIL                   : BOOL:=FALSE;
	//hardware
	fbErrorSystem:FB_ErrorSystem;
	fb_s2_EL1809:EL1809;
	fb_s3_EL1809:EL1809;
	fb_s4_EL2819:EL2819;
	fb_s5_EL2819:EL2819;
	fb_s6_EL9505:EL9505;
	fb_s7_EL1252:EL1252;
	fb_s8_EL9410:EL9410;
	fb_s9_EL1252:EL1252;
	fb_s10_EL7201:EL7201;   
	fb_s11_EL7201:EL7201;
	fb_s12_EL7201:EL7201;
	fb_s13_EL3214:EL3214;
	fb_s14_EL5021:EL5021;
	fb_s15_EL6695:EL6695;
	fb_s16_EL9410:EL9410;
	fb_s17_EL2032:EL2032;
	fb_s18_EK1110:EK1110;
	fb_s19_IndraDrive:IndraDrive;
	fb_s20_IPOS8020:iPOS8020;
	fb_s21_IPOS8020:iPOS8020;
	fb_s22_IPOS8020:iPOS8020;
	
    stStatusRot:ST_STATUS_ROT;
	
	timPhaseStabilization: TON;
	timPhaseErrorOverH1: TON;
	bPhaseOKSetReset: SR;
	fActVelOld:LREAL:=0;
	fActVelOldOld:LREAL:=0;
	iRotTempertureAlarmCounter:INT:=0;
	iIndraWarningAlarmCounter:INT:=0;
    iCounter:INT:=0;
	
END_VAR

VAR_INPUT
  stHWControlX       : ST_HW_CONTROL_XYZ;
  stHWControlY       : ST_HW_CONTROL_XYZ;
  stHWControlZ       : ST_HW_CONTROL_XYZ;
  stHWControlRot     : ST_HW_CONTROL_ROT;
  stHWStatusX        : ST_HW_STATUS_XYZ;
  stHWStatusY        : ST_HW_STATUS_XYZ;
  stHWStatusZ        : ST_HW_STATUS_XYZ;
  stHwStatusRot      : ST_HW_STATUS_ROT;
  stHWStatusDev      : ST_HW_STATUS_DEV;
  stTMSInterlocks    : ST_TMS_INTERLOCKS;
  bAllowStateTransistion: BOOL;
END_VAR

// Check hardware status
ACT_1_Hardware();

// Read Bridge Terminal Inputs
TSCS_Bridge_Inputs();

// Monitor temperature
ACT_2_Temperatures();

// Monitor temperature
ACT_3_Interlocks();

// Main motor motion
ACT_4_MainDrive();

// Steppers
ACT_5_Steppers();

// Write Bridge Terminal Outputs (incl. test)
TSCS_Bridge_Diagnostic();
TSCS_Bridge_Outputs();

// Error handling
ACT_6_Error();

// Some statses Status
ACT_7_Status();

// Post exe
eTargetStateOld:=stHwStatusRot.eTargetState;

iCounter:=iCounter+1;

ACTION ACT_1_Hardware:
// Check state of hardware

// Slave 2 EL1809: General I/O, fuses...
fb_s2_EL1809(ErrorSystem:=fbErrorSystem.pErrorSystem,En:=TRUE,iTerminal_ID:=2);
stHWStatusDev.bEStopOK:=fb_s2_EL1809.bBI_1;                       // s2: ch1: emergency stop ok                 Verify: OK   
stHWStatusX.bEStopOK:=fb_s2_EL1809.bBI_1;                         // Prepare for individula Estops
stHWStatusY.bEStopOK:=fb_s2_EL1809.bBI_1;                         // Prepare for individula Estops
stHWStatusZ.bEStopOK:=fb_s2_EL1809.bBI_1;                         // Prepare for individula Estops
stHWStatusRot.bEStopOK:=fb_s2_EL1809.bBI_1;                       // Prepare for individula Estops

stHwStatusRot.bMainDriveThermalFilterOK:=fb_s2_EL1809.bBI_2;      // s2: ch2: rf02 termal braking filter OK..   Verify: Q to Markus: Maybe this should be rd02?
stHWStatusDev.bTA01_TA02_24VSupplyOK:=fb_s2_EL1809.bBI_3;         // s2: ch3: ta01 and ta02 24V power supply OK Verify: OK  
stHWStatusDev.bFC11_Fuse24VOK:=fb_s2_EL1809.bBI_4;                // s2: ch4: fc11 24V fuse OK                   Verify: OK
stHWStatusDev.bFA01_FA02_OvervoltageOK:=fb_s2_EL1809.bBI_5;       // s2: ch5: fa01 and fa02 overvoltage protection OK
stHwStatusRot.bFuseMainRotationOK:=fb_s2_EL1809.bBI_6;            // s2: ch6: fc01 fuse target wheel motor OK
stHWStatusDev.bFC06_FC07_FuseICSOutletsOK:=fb_s2_EL1809.bBI_7;    // s2: ch7: fc06 and fc07 ICS outlets fuse OK
stHWStatusDev.bFC51_FC52_FC53_FuseUPSOK:=fb_s2_EL1809.bBI_8;      // s2: ch8: fc51, fc52 and fc53 UPS fuses OK (something wrong)

// Slave 3 EL1809: Motion switches (limits)
fb_s3_EL1809(ErrorSystem:=fbErrorSystem.pErrorSystem,En:=TRUE,iTerminal_ID:=3);
main.stHWStatusX.bLimitMax :=fb_s3_EL1809.bBI_1;          // s3: ch1: w02.bg01 stepper x limit max
main.stHWStatusX.bLimitMin :=fb_s3_EL1809.bBI_2;          // s3: ch2: w02.bg02 stepper x limit min
main.stHWStatusX.bLimitMaxMax :=fb_s3_EL1809.bBI_3;       // s3: ch3: w02.bg03 stepper x limit max max
main.stHWStatusX.bLimitMinMin :=fb_s3_EL1809.bBI_4;       // s3: ch4: w02.bg04 stepper x limit min min
main.stHWStatusY.bLimitMax :=fb_s3_EL1809.bBI_5;          // s3: ch5: w02.bg05 stepper y limit max
main.stHWStatusY.bLimitMin :=fb_s3_EL1809.bBI_6;          // s3: ch6: w02.bg06 stepper y limit min
main.stHWStatusY.bLimitMaxMax :=fb_s3_EL1809.bBI_7;       // s3: ch7: w02.bg07 stepper y limit max max
main.stHWStatusY.bLimitMinMin :=fb_s3_EL1809.bBI_8;       // s3: ch8: w02.bg08 stepper y limit min min
main.stHWStatusZ.bLimitMax :=fb_s3_EL1809.bBI_9;          // s3: ch9: w03.bg01 stepper z limit max
main.stHWStatusZ.bLimitMin :=fb_s3_EL1809.bBI_10;         // s3: ch10: w03.bg02 stepper z limit min
main.stHWStatusZ.bLimitMinPark :=fb_s3_EL1809.bBI_11;     // s3: ch11: w03.bg03 stepper z limit min service (lowest switch)
main.stHWStatusZ.bLimitMaxMax :=fb_s3_EL1809.bBI_12;      // s3: ch12: w03.bg04 stepper z limit max max
main.stHWStatusZ.bLimitMinMin :=fb_s3_EL1809.bBI_13;      // s3: ch13: w03.bg05 stepper z limit min min
main.stHWStatusZ.bLimitMinMinPark :=fb_s3_EL1809.bBI_14;  // s3: ch14: w03.bg06 stepper z limit min min service (lowest switch)
main.stHWStatusX.bLimitMinPark:=FALSE;                    // Not used
main.stHWStatusX.bLimitMinMinPark:=FALSE;                 // Not used
main.stHWStatusX.bParkingRangeEnabled:=FALSE;             // Not used;
main.stHWStatusY.bLimitMinPark:=FALSE;                    // Not used
main.stHWStatusY.bLimitMinMinPark:=FALSE;                 // Not used
main.stHWStatusY.bParkingRangeEnabled:=FALSE;             // Not used;

// Slave 4 EL2809: Feed sensors
fb_s4_EL2819(ErrorSystem:=fbErrorSystem.pErrorSystem,En:=TRUE,iTerminal_ID:=4);
stHWControlRot.bRotOmronSensor1Feed:=TRUE;     // s4: ch1: Feed omron sensor 1
stHWControlRot.bRotOmronSensor2Feed:=TRUE;     // s4: ch2: Feed omron sensor 2

// Slave 5 EL2809: Feed switches and brakes
fb_s5_EL2819(ErrorSystem:=fbErrorSystem.pErrorSystem,En:=TRUE,iTerminal_ID:=5);
stHWControlX.bMinMaxFeed:=TRUE;           // s5: ch1: kf05: w02.bg01 w02.bg02 stepper x limit switch max, limit min
//stHWControl.bXBrakeReleaseCmd           // s5: ch2: kf05: w02.ql1: stepper x brake
stHWControlX.bMinMinMaxMaxFeed:=TRUE;     // s5: ch3: kf05: w02.bg03 w02.bg04 stepper x limit switch max max, limit min min
stHWControlY.bMinMaxFeed:=TRUE;           // s5: ch5: kf05: w02.bg05 w02.bg06 stepper y limit switch max, limit min
//stHWControl.bYBrakeReleaseCmd           // s5: ch6: kf05: w02.ql2: stepper y brake
stHWControlY.bMinMinMaxMaxFeed:=TRUE;     // s5: ch7: kf05: w02.bg07 w02.bg08 stepper y limit switch max max, limit min min
stHWControlZ.bMinMaxFeed:=TRUE;           // s5: ch9: kf05: w03.bg01 w03.bg02 w03.bg03  stepper z limit switch max, limit min limit min min (service)
stHWControlZ.bMinMinMaxMaxFeed:=TRUE;     // s5: ch10: kf05: w03.bg04 w03.bg05 w03.bg06  stepper z limit switch max max, limit min min
// Note brakes needs control!!!

// s6: 5V power supply
fb_s6_EL9505(ErrorSystem:=fbErrorSystem.pErrorSystem,En:=TRUE,iTerminal_ID:=6);

// s7: time stamped 5V input from timing system (timing reference pulse 14Hz)
// s7: ch1: kf06. Timing system ref pulse (14Hz). Synch pulse ICS.
fb_s7_EL1252(ErrorSystem:=fbErrorSystem.pErrorSystem,En:=TRUE,iTerminal_ID:=7);

// s8: 24V power supply
fb_s8_EL9410(ErrorSystem:=fbErrorSystem.pErrorSystem,En:=TRUE,iTerminal_ID:=8);

// s9: Omron time stamp 24V
// s9: ch1: w01.bg01 fibre sensor input (home or sector?)
// s9: ch2: w01.bg02 fibre sensor input (home or sector?)
fb_s9_EL1252(ErrorSystem:=fbErrorSystem.pErrorSystem,En:=TRUE,iTerminal_ID:=9);

// s10 ch1: kf09 w02.bg21 Resolver X  
fb_s10_EL7201(ErrorSystem:=fbErrorSystem.pErrorSystem,En:=TRUE,iTerminal_ID:=10);

// s11 ch1: kf10 w02.bg22 Resolver Y
fb_s11_EL7201(ErrorSystem:=fbErrorSystem.pErrorSystem,En:=TRUE,iTerminal_ID:=11);

// s11 ch1: kf11 w03.bg21 Resolver Z
fb_s12_EL7201(ErrorSystem:=fbErrorSystem.pErrorSystem,En:=TRUE,iTerminal_ID:=12);

// s13 EL3214: Temperature inputs X,Y,Z and rotation
fb_s13_EL3214(ErrorSystem:=fbErrorSystem.pErrorSystem,En:=TRUE,iTerminal_ID:=13);
stHWStatusX.fStepperTemp:=INT_TO_LREAL(fb_s13_EL3214.iAI_1)/10; // s13: ch1: kf12 w02.bt01 temperature stepper X PT100
stHWStatusY.fStepperTemp:=INT_TO_LREAL(fb_s13_EL3214.iAI_2)/10; // s13: ch2: kf12 w02.bt02 temperature stepper Y PT100
stHWStatusZ.fStepperTemp:=INT_TO_LREAL(fb_s13_EL3214.iAI_3)/10; // s13: ch3: kf12 w03.bt01 temperature stepper Z PT100
stHWStatusRot.fRotTemp:=INT_TO_LREAL(fb_s13_EL3214.iAI_4)/10;   // s13: ch4: kf12 Target Main motor Temperature (KTY) (in deg*10)

// s14: Extra encoder (main rotation)
fb_s14_EL5021(ErrorSystem:=fbErrorSystem.pErrorSystem,En:=TRUE,iTerminal_ID:=14);

// s15: Communication to monitoring system
fb_s15_EL6695(ErrorSystem:=fbErrorSystem.pErrorSystem,En:=TRUE,iTerminal_ID:=15);

// s15: 24V power supply
fb_s16_EL9410(ErrorSystem:=fbErrorSystem.pErrorSystem,En:=TRUE,iTerminal_ID:=16);

// s17: MPS com.
fb_s17_EL2032(ErrorSystem:=fbErrorSystem.pErrorSystem,En:=TRUE,iTerminal_ID:=17);

// s1?: Two EL2612 Relay for MPS not in system yet
// s1?: ch1: kf17 Ready for beam
// s1?: ch2: kf17 Beam permit
// s1?: ch3: kf18 Ready for beam
// s1?: ch4: kf18 Beam permit

// s18: extension to drives
fb_s18_EK1110(ErrorSystem:=fbErrorSystem.pErrorSystem,En:=TRUE,iTerminal_ID:=18);

// s19: Main target drive
fb_s19_IndraDrive(ErrorSystem:=fbErrorSystem.pErrorSystem,En:=TRUE,iTerminal_ID:=19);

// s20: Stepper 1
fb_s20_IPOS8020(ErrorSystem:=fbErrorSystem.pErrorSystem,En:=TRUE,iTerminal_ID:=20);

// s21: Stepper 2
fb_s21_IPOS8020(ErrorSystem:=fbErrorSystem.pErrorSystem,En:=TRUE,iTerminal_ID:=21);

// s22: Stepper 3
fb_s22_IPOS8020(ErrorSystem:=fbErrorSystem.pErrorSystem,En:=TRUE,iTerminal_ID:=22);

fbErrorSystem(En:=TRUE);
END_ACTION

ACTION ACT_2_Temperatures:
// Function: Monitor tempertures
// Interlock motion on temperatures
// Author: Anders Sandström 2019

stHwStatusRot.fActTemp:=fb_s13_EL3214.iAI_4/10.0;

// Motor Temperature Monitoring Interlock (needs to be error for 1 second before trip)
IF (stHwStatusRot.fActTemp >= GVL_Parameters.nMaxMotorTemperature) THEN
    // Error for 1000 cycles in a row
	IF iRotTempertureAlarmCounter>1000 THEN
	  stHWControlRot.bEnable:= FALSE;
	  stHWControlRot.bExecute:= FALSE;
	  stHwStatusRot.nErrorId:=GVL_ErrorCodes.nErrorIndraTempToHigh;
	  stHwStatusRot.sErrorStr:=GVL_ErrorCodes.sErrorIndraTempToHigh;
    ELSE
	  iRotTempertureAlarmCounter:=iRotTempertureAlarmCounter+1; 
	END_IF
ELSE
	// reset filter
	iRotTempertureAlarmCounter:=0; // Used as filter for alarm
END_IF
END_ACTION

ACTION ACT_3_Interlocks:
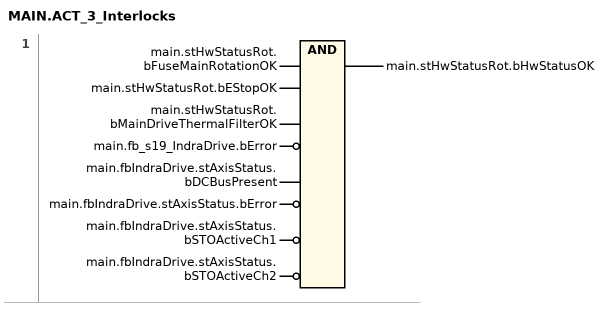
// NETWORK 1
main.stHwStatusRot.bHwStatusOK := main.stHwStatusRot.bFuseMainRotationOK AND main.stHwStatusRot.bEStopOK AND main.stHwStatusRot.bMainDriveThermalFilterOK AND NOT main.fb_s19_IndraDrive.bError AND main.fbIndraDrive.stAxisStatus.bDCBusPresent AND NOT main.fbIndraDrive.stAxisStatus.bError AND NOT main.fbIndraDrive.stAxisStatus.bSTOActiveCh1 AND NOT main.fbIndraDrive.stAxisStatus.bSTOActiveCh2;

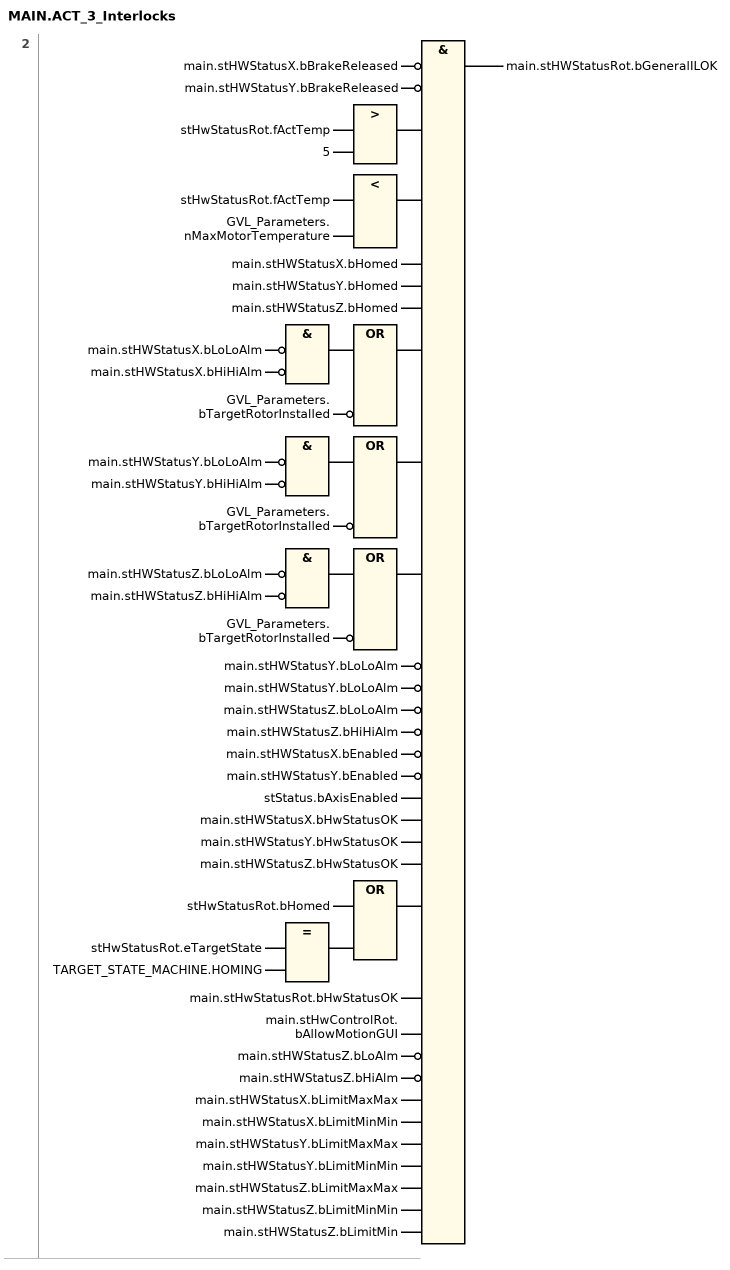
// NETWORK 2
main.stHWStatusRot.bGeneralILOK := NOT main.stHWStatusX.bBrakeReleased AND NOT main.stHWStatusY.bBrakeReleased AND stHwStatusRot.fActTemp > 5 AND stHwStatusRot.fActTemp < GVL_Parameters.nMaxMotorTemperature AND main.stHWStatusX.bHomed AND main.stHWStatusY.bHomed AND main.stHWStatusZ.bHomed AND (NOT main.stHWStatusX.bLoLoAlm AND NOT main.stHWStatusX.bHiHiAlm OR NOT GVL_Parameters.bTargetRotorInstalled) AND (NOT main.stHWStatusY.bLoLoAlm AND NOT main.stHWStatusY.bHiHiAlm OR NOT GVL_Parameters.bTargetRotorInstalled) AND (NOT main.stHWStatusZ.bLoLoAlm AND NOT main.stHWStatusZ.bHiHiAlm OR NOT GVL_Parameters.bTargetRotorInstalled) AND NOT main.stHWStatusY.bLoLoAlm AND NOT main.stHWStatusY.bLoLoAlm AND NOT main.stHWStatusZ.bLoLoAlm AND NOT main.stHWStatusZ.bHiHiAlm AND NOT main.stHWStatusX.bEnabled AND NOT main.stHWStatusY.bEnabled AND stStatus.bAxisEnabled AND main.stHWStatusX.bHwStatusOK AND main.stHWStatusY.bHwStatusOK AND main.stHWStatusZ.bHwStatusOK AND (stHwStatusRot.bHomed OR stHwStatusRot.eTargetState = TARGET_STATE_MACHINE.HOMING) AND main.stHwStatusRot.bHwStatusOK AND main.stHwControlRot.bAllowMotionGUI AND NOT main.stHWStatusZ.bLoAlm AND NOT main.stHWStatusZ.bHiAlm AND main.stHWStatusX.bLimitMaxMax AND main.stHWStatusX.bLimitMinMin AND main.stHWStatusY.bLimitMaxMax AND main.stHWStatusY.bLimitMinMin AND main.stHWStatusZ.bLimitMaxMax AND main.stHWStatusZ.bLimitMinMin AND main.stHWStatusZ.bLimitMin;

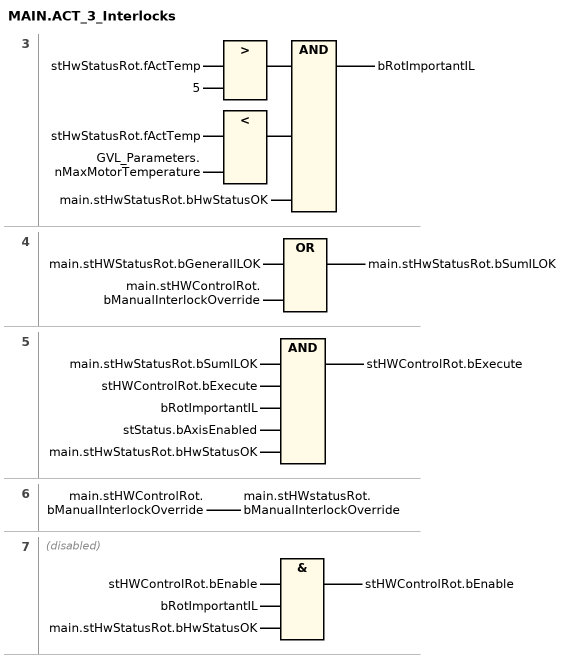
// NETWORK 3
bRotImportantIL := stHwStatusRot.fActTemp > 5 AND stHwStatusRot.fActTemp < GVL_Parameters.nMaxMotorTemperature AND main.stHwStatusRot.bHwStatusOK;

// NETWORK 4
main.stHwStatusRot.bSumILOK := main.stHWStatusRot.bGeneralILOK OR main.stHWControlRot.bManualInterlockOverride;

// NETWORK 5
stHWControlRot.bExecute := main.stHwStatusRot.bSumILOK AND stHWControlRot.bExecute AND bRotImportantIL AND stStatus.bAxisEnabled AND main.stHwStatusRot.bHwStatusOK;

// NETWORK 6
main.stHWstatusRot.bManualInterlockOverride := main.stHWControlRot.bManualInterlockOverride;

// NETWORK 7 (disabled)
// stHWControlRot.bEnable := stHWControlRot.bEnable AND bRotImportantIL AND main.stHwStatusRot.bHwStatusOK;
END_ACTION

ACTION ACT_4_MainDrive:

// Enable Axis independent of state (Ensure that drive is ready to enable)
IF stHWControlRot.bEnable THEN
   IF stStatus.bDCBusPresent AND NOT stStatus.bSTOActiveCh1 AND NOT stStatus.bSTOActiveCh2 AND NOT stStatus.bError AND main.stHwStatusRot.bHwStatusOK THEN 
	   // Everything is OK, allow enable of drive.
      stCommands.bEnableAxis :=stHWControlRot.bEnable;
   ELSE
	   // Something is not right.. STO, hardware...
	   stCommands.bEnableAxis := FALSE;
	   stHWControlRot.bExecute := FALSE;
	   stHwStatusRot.bError:=TRUE;
	   stHwStatusRot.nErrorId:=GVL_ErrorCodes.nErrorIndraNotReady;
	   stHwStatusRot.sErrorStr:=GVL_ErrorCodes.sErrorIndraNotReady; 
   END_IF
ELSE
	//Reset enable
    stCommands.bEnableAxis:=stHWControlRot.bEnable;
END_IF

// filter bWarning otherwsie it will trip on each positive edge of bExecute
IF fbIndraDrive.stAxisStatus.bWarning  AND iIndraWarningAlarmCounter<100 THEN
	iIndraWarningAlarmCounter:=iIndraWarningAlarmCounter+1;
ELSIF NOT fbIndraDrive.stAxisStatus.bWarning THEN
	iIndraWarningAlarmCounter:=0;	
END_IF

// Alarm and stop on prewarning
IF iIndraWarningAlarmCounter>=99 AND fbIndraDrive.stAxisStatus.nDiagMessage=-1072816047  THEN
  stHwStatusRot.nErrorId:=GVL_ErrorCodes.nErrorIndraOverHeatPrewarning;
  stHwStatusRot.sErrorStr:=GVL_ErrorCodes.sErrorIndraOverHeatPrewarning; 
  stCommands.bEnableAxis := FALSE;
  stHWControlRot.bExecute := FALSE;
ELSIF iIndraWarningAlarmCounter>=99 THEN
  //Only warning
  stHwStatusRot.nErrorId:=GVL_ErrorCodes.nErrorIndraWarning;
  stHwStatusRot.sErrorStr:=GVL_ErrorCodes.sErrorIndraWarning;
  stCommands.bEnableAxis := FALSE;
  stHWControlRot.bExecute := FALSE; 
END_IF

// Take down enable if STO
IF stStatus.bSTOActiveCh1 OR stStatus.bSTOActiveCh2 THEN
	stCommands.bEnableAxis:=FALSE;
	stHWControlRot.bEnable:=FALSE;
	stHWControlRot.bExecute:=FALSE;
END_IF

IF stHWControlRot.bExecute THEN
  IF stStatus.bAxisEnabled THEN
	// Axis enabled so execute command
    stCommands.bHaltAxis:=stHWControlRot.bExecute;
  ELSE
	 // Axis not enabled so reset bExecute and issue an error
	stHWControlRot.bExecute:=FALSE;
	stCommands.bHaltAxis:=FALSE;
	stHwStatusRot.bError:=TRUE;
	stHwStatusRot.nErrorId:=GVL_ErrorCodes.nErrorNotEnabled;
	stHwStatusRot.sErrorStr:=GVL_ErrorCodes.sErrorNotEnabled; 
  END_IF
ELSE
  stCommands.bHaltAxis:=stHWControlRot.bExecute;
END_IF

// Always reset (probbaly not needed since above if statement)
IF NOT stCommands.bEnableAxis THEN
  stHWControlRot.bExecute:=FALSE;
END_IF

// Status to EPICS
stHwStatusRot.bEnabled:=stStatus.bAxisEnabled;
stCommands.bCmd_ErrorReset:=stHWControlRot.bReset;

// Do not allow drive controlled homing
stCommands.bCmd_DriveControlledHoming:=FALSE;

// State change allow change from CONST velo to Phase and back
bAllowStateTransistion:=FALSE;

IF (stHWControlRot.eTargetStateCmd = TARGET_STATE_MACHINE.PHASING OR 
    stHWControlRot.eTargetStateCmd = TARGET_STATE_MACHINE.CONSTANT_VELOCITY) AND 
    (stHwStatusRot.eTargetState = TARGET_STATE_MACHINE.PHASING OR 
    stHwStatusRot.eTargetState = TARGET_STATE_MACHINE.CONSTANT_VELOCITY)
 THEN
	bAllowStateTransistion:=TRUE;
END_IF

// Do not allow to go to POSITION mode (and other modes) while running
IF stHWControlRot.eTargetStateCmd <> stHwStatusRot.eTargetState AND (NOT 
    stHWControlRot.bexecute AND 
    stStatus.bAxisStandStillStatus) OR bAllowStateTransistion THEN
    stHwStatusRot.eTargetState:=stHWControlRot.eTargetStateCmd;
END_IF

// Ensure valid phase offset
IF stHWControlRot.fPhaseOffsetMM > GVL_Parameters.fMaxPhaseOffsetMM THEN
	stHWControlRot.fPhaseOffsetMM :=  GVL_Parameters.fMaxPhaseOffsetMM;
END_IF
IF stHWControlRot.fPhaseOffsetMM < GVL_Parameters.fMinPhaseOffsetMM THEN
	stHWControlRot.fPhaseOffsetMM :=  GVL_Parameters.fMinPhaseOffsetMM;
END_IF

stHwStatusRot.fPhaseOffsetActDeg := stHWControlRot.fPhaseOffsetMM /(GVL_Parameters.fWheelDiameter*pi/360.0);

//To high velo?
IF ABS(stHWControlRot.fVelSet) > GVL_Parameters.fMaximumSPeedSPRpm  OR 
  (ABS(stHwStatusRot.fActVel) > GVL_Parameters.fMaximumSPeedRpm  AND ABS(fActVelOld) >  GVL_Parameters.fMaximumSPeedRpm AND 
   ABS(fActVelOldOld) >  GVL_Parameters.fMaximumSPeedRpm) THEN
	stHWControlRot.fVelSet:=0;
	stHWControlRot.bEnable:=0;
	stHWControlRot.bExecute:=0;
	stHwStatusRot.bError:=TRUE;
	stHwStatusRot.nErrorId:=GVL_ErrorCodes.nErrorVelToHigh;
	stHwStatusRot.sErrorStr:=GVL_ErrorCodes.sErrorVelToHigh;
END_IF

//nAdditiveTorqueSetpoint:=0;
//IF NOT  stHWControlRot.bExecute THEN
//	addStartupTorqueTrigger:=TRUE;
//END_IF

// Clear homed bit if drive is re-parametrizied or lost connection
IF stStatus.bDriveInParameterMode OR MAIN.fb_s19_IndraDrive.InfoData_State <> 8 THEN
	stHwStatusRot.bHomed:=FALSE;
	stHWControlRot.fVelSet:=0;
	stHWControlRot.bEnable:=0;
	stHWControlRot.bExecute:=0;
	stHwStatusRot.bError:=TRUE;
	stHwStatusRot.nErrorId:=GVL_ErrorCodes.nErrorNeedHoming;
	stHwStatusRot.sErrorStr:=GVL_ErrorCodes.sErrorNeedHoming;
END_IF

// Calculate actual velcoity based on latched positions from timing system (distance since last latch divided with 71ms).
// Only calculate if over 3rpm
fbCalcVeloLatch(
            fVeloLimit:=3,
			dLatchedPosition:= dLatchedPosition);

// Run the current requested mode. The modes are:
//  * CONSTANT_VELOCITY : Run wheel at a constant velocity
//  * POSITION          : Positions the wheel at a certain angle
//  * PHASE             : Control phase of wheel (normal "production" state/mode) 
//  * HOMING            : Runs homing sequence to reference rotational encoder 
//                        based on encoder ring ref mark. Then apply offset.
//  * TORQUE            : Apply constant torque. This mode is NOT USED, only for testing.
CASE stHwStatusRot.eTargetState OF 
	TARGET_STATE_MACHINE.CONSTANT_VELOCITY:
        stCommands.fCommandAcceleration:=GVL_Parameters.fAccDefaultVel;
        stCommands.fCommandDeceleration:=GVL_Parameters.fAccDefaultVel;
		fbModeVelo(
            bExecute:=         stHWControlRot.bExecute,
            bReset:=           stHWControlRot.bReset,
			fVelSet:=          stHWControlRot.fVelSet,
			stStatus:=	       stStatus,	
			stCommands:=       stCommands);
			
			//ramp velocity with selected acceleration
			fbRampVelo(bExecute:=stHWControlRot.bExecute,
              fVelSetIn:=fbModeVelo.fSpeedSetpoint,
              iBlockSampleTimeMicroS:=GVL_Parameters.nTaskSampleTime*1000,
              fVelSetOut:=stCommands.fVelocityCommandValue,
              fVelActIn:=stStatus.fActualVelocity/10);
			  
// add extra torque att startup TEST
		//	IF stStatus.bAxisEnabled AND stHWControlRot.bExecute AND stHWControlRot.fVelSet > 0 THEN
		//		IF stStatus.fActualVelocity/10< stHWControlRot.fVelSet/2 THEN
		//	        nAdditiveTorqueSetpoint:=100;  //Add 10% when under x rpm
		//		ELSIF stStatus.fActualVelocity/10 > stHWControlRot.fVelSet/2 THEN
		//			nAdditiveTorqueSetpoint:=40;
		//		END_IF
		//	END_IF

			
	TARGET_STATE_MACHINE.POSITIONING:
	    stCommands.fCommandAcceleration:=GVL_Parameters.fAccDefaultPos;
        stCommands.fCommandDeceleration:=GVL_Parameters.fAccDefaultPos;

		fbModePos(
            bExecute:=         stHWControlRot.bExecute,
            bReset:=           stHWControlRot.bReset,
			fVelSet:=          stHWControlRot.fVelSet,
			fPosSet:=          stHWControlRot.fPosSet,
			fRefOffset:=       fbModeHome.fActPositionOffset,
			stStatus:=         stStatus,	
			stCommands:=       stCommands);
		
	TARGET_STATE_MACHINE.PHASING:
	    stCommands.fCommandAcceleration:=GVL_Parameters.fAccDefaultVel;
        stCommands.fCommandDeceleration:=GVL_Parameters.fAccDefaultVel;
   		fbModePhase(
			bExecute:=         stHWControlRot.bExecute,
            bReset:=           stHWControlRot.bReset,
			stStatus:=	       stStatus,
			dLatchedPosition:= dLatchedPosition,
			ePhaseType:=       stHWControlRot.ePhaseCntrlAlg,
			ePwmType:=         stHWControlRot.ePhasePwmType,
			stCommands:=       stCommands,
            fPhaseOffsetMM:=   stHWControlRot.fPhaseOffsetMM,
            fRefOffset:=       fbModeHome.fActPositionOffset);
			
			//ramp velocity with selected acceleration (as long as not phasing)
			IF NOT fbModePhase.bPhasing THEN
              fbRampVelo(bExecute:=stHWControlRot.bExecute,
                fVelSetIn:=fbModePhase.fSpeedSetpoint,
                iBlockSampleTimeMicroS:=GVL_Parameters.nTaskSampleTime*1000,
                fVelSetOut:=stCommands.fVelocityCommandValue,
                fVelActIn:=fbModePhase.fLastSectorVelocity);
			ELSE // if phasing then take setpoint direct from fbModePhase
			  stCommands.fVelocityCommandValue:=fbModePhase.fSpeedSetpoint;
            END_IF
						
	TARGET_STATE_MACHINE.HOMING:
        stCommands.fCommandAcceleration:=GVL_Parameters.fAccDefaultVel;
        stCommands.fCommandDeceleration:=GVL_Parameters.fAccDefaultVel;
        fbModeHome( 
            bExecute:=         stHWControlRot.bExecute,
            bReset:=           stHWControlRot.bReset,
			bHomed:=           stHwStatusRot.bHomed,
			fVelSet:=          GVL_Parameters.fHomeSpeedRpm,
			fPosSet:=          stHWControlRot.fPosSet,
			stStatus:=	       stStatus,	
			stCommands:=       stCommands);
		//stCommands.fFeedrateOverride:=1.0;
		//ramp velocity with selected acceleration
		fbRampVelo(bExecute:=stHWControlRot.bExecute,
              fVelSetIn:=fbModeHome.fSpeedSetpoint,
              iBlockSampleTimeMicroS:=GVL_Parameters.nTaskSampleTime*1000,
              fVelSetOut:=stCommands.fVelocityCommandValue,
              fVelActIn:=stStatus.fActualVelocity/10);
 
	TARGET_STATE_MACHINE.TORQUE:
	    stCommands.fCommandAcceleration:=GVL_Parameters.fAccDefaultVel;
        stCommands.fCommandDeceleration:=GVL_Parameters.fAccDefaultVel;
		stCommands.eOperationMode:=E_OPERATION_MODE_NO.eSecondaryOpMode7;
	    stCommands.eMotionMode :=e_Motion_mode.eJogPositive;
	
	  ELSE  // No valid state
		bApplyTorqueFF:=FALSE;
		stHWControlRot.bExecute:=FALSE;
        stHWControlRot.bEnable:=FALSE;
		stCommands.fVelocityCommandValue:=0;
		stCommands.fCommandVelocity:=0;
		stCommands.fCommandAcceleration:=0;
        stCommands.fCommandDeceleration:=0;
		stHwStatusRot.nErrorId:=GVL_ErrorCodes.nErrorInvalidState;
	    stHwStatusRot.sErrorStr:=GVL_ErrorCodes.sErrorInvalidState;
END_CASE

// This code is kept in case a need for applying a feedforward torque is ever needed. Then this is a good example.
(*IF bApplyTorqueFF THEN
  // add extra torque att startup TEST
  IF stStatus.bAxisEnabled AND stHWControlRot.bExecute(*AND stHWControlRot.bExecute*) THEN
	 //Positive
	IF stCommands.fVelocityCommandValue >= GVL_Parameters.fMinVelSetpointAbsRpm THEN
	   IF stStatus.fActualVelocity/10 > GVL_Parameters.fMinVelSetpointAbsRpm THEN
	     nAdditiveTorqueSetpoint:=LREAL_TO_INT(GVL_Parameters.fNominalFFTourqueAbs*10);
	   ELSIF stStatus.fActualVelocity/10 < GVL_Parameters.fMinVelSetpointAbsRpm/10 THEN  // Add more tourqe at startup
		 nAdditiveTorqueSetpoint:=LREAL_TO_INT(GVL_Parameters.fStartupFFTourqueAbs*10);
	   END_IF
	ELSIF  stCommands.fVelocityCommandValue <= -GVL_Parameters.fMinVelSetpointAbsRpm THEN
		IF stStatus.fActualVelocity/10 < -GVL_Parameters.fMinVelSetpointAbsRpm THEN
	      nAdditiveTorqueSetpoint:=-LREAL_TO_INT(GVL_Parameters.fNominalFFTourqueAbs*10);
	    ELSIF  stStatus.fActualVelocity/10 > -GVL_Parameters.fMinVelSetpointAbsRpm/10 THEN // Add more tourqe at startup
		  nAdditiveTorqueSetpoint:=-LREAL_TO_INT(GVL_Parameters.fStartupFFTourqueAbs*10);
	   END_IF
    END_IF
  ELSE
    nAdditiveTorqueSetpoint:=0;
  END_IF
ELSE
  nAdditiveTorqueSetpoint:=0;
END_IF*)
// Force feedforward setpoint to 0 since not used.
nAdditiveTorqueSetpoint:=0;

// Stop if not bExecute
IF NOT stHWControlRot.bExecute THEN
	stCommands.fVelocityCommandValue:=0;
END_IF

// Check maximum velocity (Ensure velocity command is not higher than allowed)
IF stCommands.fCommandVelocity > GVL_Parameters.fMaximumSPeedRpm THEN
  stCommands.fCommandVelocity := GVL_Parameters.fMaximumSPeedRpm;
END_IF
IF stCommands.fVelocityCommandValue > GVL_Parameters.fMaximumSPeedRpm THEN
  stCommands.fVelocityCommandValue := GVL_Parameters.fMaximumSPeedRpm;
END_IF

// Run Rexroth  communication FB.
// Note: This FB is from rexroth but a few fixes/changes have been added
fbIndraDrive(
	AmsNetId:= stAmsNetId, 
	AdsAddr_Port:= nPort, 
	stAxisCommands:= stCommands, 
	stDriveStatus:= , 
	stAxisStatus=> stStatus, 
	stDriveCommands=> );

// Calculate values for status in EPICS
stHwStatusRot.fSetVelRaw:= DINT_TO_LREAL(MAIN.fbIndraDrive.stDriveCommands.nS40_VelocityCommandValue)/10000;	
stHwStatusRot.fActPos:=stStatus.fActualPosition-fbModeHome.fActPositionOffset;
IF stHwStatusRot.fActPos > 360 THEN
  stHwStatusRot.fActPos:=stHwStatusRot.fActPos-360;	
END_IF
IF stHwStatusRot.fActPos < 0 THEN
  stHwStatusRot.fActPos:=stHwStatusRot.fActPos+360;	
END_IF
stHwStatusRot.fActTorque:=stStatus.fActualTorque;
fActVelOldOld:=fActVelOld;
fActVelOld:=stHwStatusRot.fActVel;
stHwStatusRot.fActVel:=stStatus.fActualVelocity/10;

// Ensure torque is not higher that allowed
stCommands.fTorqueLimit:=GVL_Parameters.fMaxRotationBipolarTorque; //%
END_ACTION

ACTION ACT_5_Steppers:
// NOT USED ANYMORE
// Motion of steppers handled in PRG "MAIN_NORMAL_MOTION"
END_ACTION

ACTION ACT_6_Error:
// Function: Error handling
// Author: Anders Sandström 2019
// Check errors of all rotational FB:s
IF stHwStatusRot.eTargetState = TARGET_STATE_MACHINE.PHASING THEN
  IF fbModePhase.bError AND NOT stHwStatusRot.bError THEN
	stHwStatusRot.bError:=fbModePhase.bError;
	stHwStatusRot.nErrorId:=fbModePhase.nErrorId;
	stHwStatusRot.sErrorStr:=fbModePhase.sErrorStr;
  END_IF
  
ELSIF stHwStatusRot.eTargetState = TARGET_STATE_MACHINE.CONSTANT_VELOCITY THEN
  IF fbModeVelo.bError AND NOT stHwStatusRot.bError THEN
	stHwStatusRot.bError:=fbModeVelo.bError;
	stHwStatusRot.nErrorId:=fbModeVelo.nErrorId;
	stHwStatusRot.sErrorStr:=fbModeVelo.sErrorStr;
  END_IF
  
ELSIF stHwStatusRot.eTargetState = TARGET_STATE_MACHINE.POSITIONING THEN
  IF fbModePos.bError AND NOT stHwStatusRot.bError THEN
	stHwStatusRot.bError:=fbModePos.bError;
	stHwStatusRot.nErrorId:=fbModePos.nErrorId;
	stHwStatusRot.sErrorStr:=fbModePos.sErrorStr;
  END_IF
  
ELSIF stHwStatusRot.eTargetState = TARGET_STATE_MACHINE.HOMING THEN
  IF fbModeHome.bError AND NOT stHwStatusRot.bError THEN
    stHwStatusRot.bError:=fbModeHome.bError;
	stHwStatusRot.nErrorId:=fbModeHome.nErrorId;
	stHwStatusRot.sErrorStr:=fbModeHome.sErrorStr;
  END_IF
END_IF

IF stHWControlRot.bReset THEN
  stHwStatusRot.bError:=FALSE;
  stHwStatusRot.nErrorId:=GVL_ErrorCodes.nErrorCodeOKId;
  stHwStatusRot.sErrorStr:=GVL_ErrorCodes.nErrorCodeOKStr;
  stHwStatusRot.bBrake1TempAlarm:=FALSE;
  stHwStatusRot.bBrake2TempAlarm:=FALSE;
  GVL.astAxes[1].stControl.bReset:=NOT(GVL.astAxes[1].stControl.bReset);
  GVL.astAxes[2].stControl.bReset:=NOT(GVL.astAxes[2].stControl.bReset);
  GVL.astAxes[3].stControl.bReset:=NOT(GVL.astAxes[3].stControl.bReset);
  iIndraWarningAlarmCounter:=0;
END_IF
//stHWControlRot.bReset:=FALSE;
END_ACTION

ACTION ACT_7_Status:
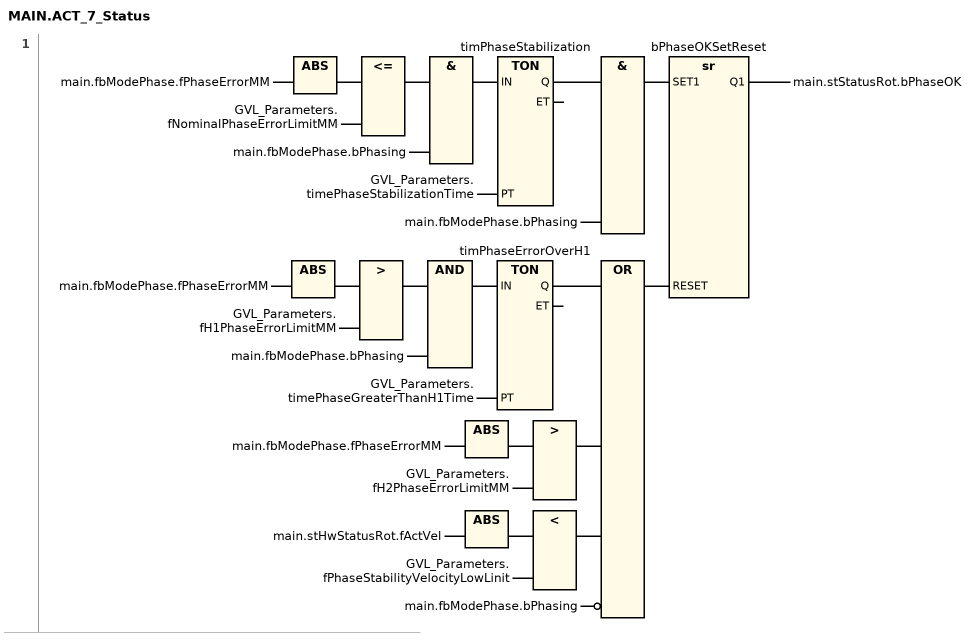
// NETWORK 1
timPhaseStabilization(IN := ABS(main.fbModePhase.fPhaseErrorMM) <= GVL_Parameters.fNominalPhaseErrorLimitMM AND main.fbModePhase.bPhasing, PT := GVL_Parameters.timePhaseStabilizationTime); // TON
timPhaseErrorOverH1(IN := ABS(main.fbModePhase.fPhaseErrorMM) > GVL_Parameters.fH1PhaseErrorLimitMM AND main.fbModePhase.bPhasing, PT := GVL_Parameters.timePhaseGreaterThanH1Time); // TON
bPhaseOKSetReset(SET1 := timPhaseStabilization.Q AND main.fbModePhase.bPhasing, RESET := timPhaseErrorOverH1.Q OR ABS(main.fbModePhase.fPhaseErrorMM) > GVL_Parameters.fH2PhaseErrorLimitMM OR ABS(main.stHwStatusRot.fActVel) < GVL_Parameters.fPhaseStabilityVelocityLowLinit OR NOT main.fbModePhase.bPhasing); // sr
main.stStatusRot.bPhaseOK := bPhaseOKSetReset.Q1;
END_ACTION

ACTION ACT_X_Diag:
// Function: Some parameters just for debugging
// Note: Do not need to be executed, can be watched online anyway..
// Author: Anders Sandström 2019

	stCommands.bCmd_ActivateParameterMode;//True puts the drive in parameter mode
	stCommands.bCmd_DisableLimits;// True disables monitoring of errors
	stCommands.bCmd_DriveControlledHoming;// True starts homing procedure defined in the drive
	stCommands.bCmd_ErrorReset;
	stCommands.bCmd_ExitParameterMode;
	stCommands.bCmd_RunVirtualMater;// Jog command to the virtual master
	stCommands.bCmd_SetAbsolutePosition;
	stCommands.bCommandPositionChange;// Drive moves to the current target position, when bCommandVAlueAccept toggled, drive moves to the new target position
	stCommands.bCommandValueAccept;// Used in "Drive positioning Mode" to update the target position when toggled
	stCommands.bEnableAxis;
	stCommands.bHaltAxis;// Performs halt on the drive, bEnableaxis has to be TRUE
	stCommands.bPositionCommandValue;//0=Absolute;1=Relative
	stCommands.eMotionMode;
	stCommands.eOperationMode;
	stCommands.fCommandAcceleration;// Acceleration used for positioning and jogging
	stCommands.fCommandDeceleration;// Deceleration used for positioning and jogging
	stCommands.fCommandPosition;
	stCommands.fCommandVelocity;// Velocity used for positioning and jogging
	stCommands.fFeedrateOverride;// Parameter used for adjustment of the velocity (0,100)%
	stCommands.fTorqueLimit;
	stCommands.fVelocityCommandValue;// S40, velocity used for positining and jogging (in velocity mode)
	stStatus.bAxisEnabled;
END_ACTION

END_PROGRAM

// ---- POUs/Target/FB_ModePhasing.TcPOU
FUNCTION_BLOCK FB_ModePhasing
VAR_INPUT
	bExecute           : BOOL         := FALSE;
	bReset             : BOOL         := FALSE;
	stStatus           : ST_INDRADRIVE_AXIS_STATUS;
    dLatchedPosition   : DINT         := 0;
	//fPhaseOffsetDeg    : LREAL        := 0;
    fPhaseControlKp    : LREAL        := 0.0012;
	fPhaseControlKi    : LREAL        := 0.00015;
	fPhaseControlKd    : LREAL        := 0.0;
	fPhaseControlKff   : LREAL        := 0.0;
	fPhaseOffsetMM     : LREAL        := 0.0;
	fRefOffset         : LREAL        :=0;  //Offset from homing
	bPhaseControlReset : BOOL         := FALSE;
	ePhaseType         : E_PHASE_TYPE := E_PHASE_TYPE.SUPERIMPOSE;
	ePwmType           : E_PWM_TYPE   := E_PWM_TYPE.NONE;
END_VAR
VAR_OUTPUT
	bError             : BOOL;
	nErrorId           : UDINT;
	sErrorStr          : STRING := GVL_ErrorCodes.nErrorCodeOKStr;
	bPhasing           : BOOL;
	fSpeedSetpoint     : LREAL;
END_VAR
VAR_IN_OUT
	stCommands         : ST_INDRADRIVE_AXIS_COMMAND;
END_VAR
VAR
  bNewTriggPulse           : BOOL  := FALSE;
  bExecuteSuperImpose      : BOOL  := FALSE;
  bVeloStable              : BOOL  := FALSE;
  bPhaseAlgTrigg           : BOOL  := FALSE;
  nClosestSectorId         : INT   := 0;
  nPIDExeSkipCounter       : INT   := 0;
  iFiltVeloArrayIndex      : INT   := 0;
  i                        : INT   := 0;
  iRangeOKCounter          : INT   := 0;
  iRangeOKCounterOld       : INT   := 0;
  nChoosenSector           : INT   := 0;
  dLatchedPositionOld      : DINT  := 0;
  fLatchedPositionOld      : LREAL := 0;
  fDistBetweenLastPulses   : LREAL := 0;
  fLastSectorVelocity      : LREAL := 0;
  fLatchedPosition         : LREAL := 0;
  fPhaseError              : LREAL := 0;
  fPhaseErrorFiltered      : LREAL := 0;
  fPhaseErrorMM            : LREAL := 0;
  fLastSectorVelocityOld   : LREAL := 0;
  fMaxValue                : LREAL := 0;
  fMinValue                : LREAL := 0;
  fRange                   : LREAL := 0;
  fDeltaVelo               : LREAL := 0;
  fNomSpeedSetAdjust       : LREAL := 0;
  fPidAdd                  : LREAL := 0;
  fSpeedSetpointLocal      : LREAL := 0;
  fArrayFiltVelo           : ARRAY[ 0 ..35] OF LREAL;
  fArrayPhaseErrorFilt     : ARRAY[ 0 ..99] OF LREAL;
  fbPhasePID               : FB_PID;
  fbPWM                    : FB_PWM;
  fbSuperImpose            : FB_TargetSuperImpose;
  timerCheckLatchFreqHigh  : TON;
  timerCheckLatchFreqLow   : TOF;
  nMissedTimingPulses      : INT:=0;
  nMissedTimingPulsesOld   : INT:=0;
  nMissedTimingPulsesLow   : INT:=0;
  nMissedTimingPulsesLowold : INT:=0;
END_VAR

// Function: 
// 1. Wait for stable velocity then start "phasing" (depending on ePhaseMode)
// 2. Choose sector for control
// 3. Calculate phase error (buffer several revs and filter)
// 4. Adjust velo setpoint to minimize phase error (PID)
// 5. PWM of the new velocity setpoint in order to increase resolution
// Note: Seems the indradrive can only hanlde 3 decimals (even if 4 is seen in interface and indradrive software)
// Author: Anders Sandström 2018

stCommands.fCommandDeceleration:=GVL_Parameters.fAccDefaultVel;	
stCommands.fCommandAcceleration:= GVL_Parameters.fAccDefaultVel;
stCommands.eMotionMode :=e_Motion_mode.eJogPositive;
stCommands.eOperationMode:=e_Operation_mode_no.eSecondaryOpMode2;

bNewTriggPulse:=FALSE;
bPhasing:=FALSE;
fNomSpeedSetAdjust:=GVL_Parameters.fNominalSpeedRpm + GVL_Parameters.fNominalSpeedAdjust; // Adjust speed setpoint
bPhasing:=bPhaseAlgTrigg;

// Reset alg
IF NOT bExecute OR bPhaseControlReset THEN
  bPhaseAlgTrigg:=FALSE;
END_IF

fLatchedPositionOld:=fLatchedPosition;  // Backup old
fLatchedPosition:=DINT_TO_LREAL(dLatchedPosition)/10000.0-fRefOffset;  // remove homing offset
IF fLatchedPosition > 360 THEN
  fLatchedPosition:=fLatchedPosition - 360;	
END_IF
IF fLatchedPosition < 0 THEN
  fLatchedPosition:=fLatchedPosition + 360;	
END_IF

// New trigger from timing system
IF (fLatchedPosition-fLatchedPositionOld)<>0 THEN
  IF(fLatchedPositionOld>fLatchedPosition) THEN
	fDistBetweenLastPulses:=(360-fLatchedPositionOld+fLatchedPosition);
  ELSE
	fDistBetweenLastPulses:=fLatchedPosition-fLatchedPositionOld;
  END_IF

  bNewTriggPulse:=TRUE;
  fLastSectorVelocity:=fDistBetweenLastPulses*GVL_Parameters.nPulseFreqHz*60/360;
  nClosestSectorId:= LREAL_TO_INT(fLatchedPosition/10);
  
  // Check if stable velocity (close to nominal)	
  iRangeOKCounterOld:=iRangeOKCounter;
  fArrayFiltVelo[iFiltVeloArrayIndex]:=fLastSectorVelocity;
  iFiltVeloArrayIndex:=iFiltVeloArrayIndex+1;
  IF iFiltVeloArrayIndex>35 THEN
	iFiltVeloArrayIndex:=0;
  END_IF
  fLastSectorVelocityOld:=fLastSectorVelocity;
  fMaxValue:=fArrayFiltVelo[0];
  fMinValue:=fArrayFiltVelo[0];
  FOR i:=1 TO 35 BY 1 DO
    IF fArrayFiltVelo[i]> fMaxValue THEN
	  fMaxValue:=fArrayFiltVelo[i];  
    END_IF
    IF fArrayFiltVelo[i]< fMinValue THEN
      fMinValue:=fArrayFiltVelo[i];  
    END_IF
  END_FOR;
  fRange:=fMaxValue-fMinValue;
  IF fRange < GVL_Parameters.fPhaseSpeedTol AND 
     ABS(fNomSpeedSetAdjust-fMinValue) < GVL_Parameters.fPhaseSpeedTol AND  
     ABS(fNomSpeedSetAdjust-fMaxValue) < GVL_Parameters.fPhaseSpeedTol THEN
	IF iRangeOKCounter <= GVL_Parameters.nVeloInRangeCount THEN
      iRangeOKCounter:=iRangeOKCounter+1;
	END_IF
  ELSE
	iRangeOKCounter:=0; 
  END_IF
  bVeloStable:=iRangeOKCounter >= GVL_Parameters.nVeloInRangeCount;
  IF bVeloStable AND NOT bPhaseAlgTrigg (*AND bTEst*) THEN
    nChoosenSector:=nClosestSectorId-1;
    bPhaseAlgTrigg:=TRUE;
    MEMSET(destAddr:=ADR(fArrayPhaseErrorFilt[0]),0,SIZEOF(fArrayPhaseErrorFilt));
    fPhaseErrorFiltered:=0;
  END_IF
END_IF

//Ensure that pulses arrive from timing system when velocity is above certain limit
IF ABS(stStatus.fActualVelocity/10) > GVL_Parameters.fCheckTimingPulseMinVel THEN
 
  IF timerCheckLatchFreqLow.Q AND fLatchedPosition <> fLatchedPositionOld THEN  // To early time trigger
	nMissedTimingPulsesLow:=nMissedTimingPulsesLow+1;
  END_IF
  timerCheckLatchFreqLow(IN:=fLatchedPosition <> fLatchedPositionOld,PT:=LREAL_TO_TIME(1000/GVL_Parameters.nPulseFreqHz- 5));
  timerCheckLatchFreqHigh(IN:=fLatchedPosition = fLatchedPositionOld,PT:=LREAL_TO_TIME(1000/GVL_Parameters.nPulseFreqHz + 5));
  
  IF timerCheckLatchFreqHigh.Q THEN // to late timing pulse
    nMissedTimingPulses:=nMissedTimingPulses+1;
	timerCheckLatchFreqHigh(IN:=FALSE);  //Reset
  END_IF
ELSE
  timerCheckLatchFreqHigh(IN:=FALSE);  //Reset
END_IF
  
IF NOT bPhaseAlgTrigg THEN
  fPhaseError:=nClosestSectorId*10-fLatchedPosition;
END_IF

IF bNewTriggPulse THEN
  nChoosenSector:=nChoosenSector+1;
  IF nChoosenSector > 35 THEN
    nChoosenSector:=0;
  END_IF	
END_IF

// Calculate phase error
IF bPhaseAlgTrigg THEN
  fPhaseError:=nChoosenSector*10-fLatchedPosition;
  IF fPhaseError >=180 THEN
	fPhaseError:=360-fPhaseError;
  ELSIF fPhaseError<-180 THEN
	fPhaseError:=fPhaseError+360;
  END_IF
ELSE
  fPhaseError:=nClosestSectorId*10-fLatchedPosition;
END_IF
fPhaseErrorMM:=fPhaseError*GVL_Parameters.fWheelDiameter*pi/360.0 + fPhaseOffsetMM; 

//Filter phase error
IF bNewTriggPulse THEN
  MEMMOVE(destAddr:=ADR(fArrayPhaseErrorFilt[1]),srcAddr:=ADR(fArrayPhaseErrorFilt[0]),SIZEOF(LREAL)*(GVL_Parameters.nPhaseErrorFilterSize-1));
  fArrayPhaseErrorFilt[0]:=fPhaseErrorMM;
  fPhaseErrorFiltered:=0;
  FOR i := 0 TO (GVL_Parameters.nPhaseErrorFilterSize-1) DO
    fPhaseErrorFiltered:=fPhaseErrorFiltered+fArrayPhaseErrorFilt[i];
  END_FOR
  fPhaseErrorFiltered:=fPhaseErrorFiltered/GVL_Parameters.nPhaseErrorFilterSize;
END_IF

IF NOT fbSuperImpose.bBusy  THEN
  bExecuteSuperImpose:= NOT bExecuteSuperImpose;
END_IF

// Control phase in different ways
// 1: PID
// 2: Superimpose
// 3: Only measure
CASE ePhaseType OF
  E_PHASE_TYPE.PID: 
    // Phasing using PID controller
	//  PID controller with integral anti windup is used to control phase error
	
    IF bNewTriggPulse AND bPhaseAlgTrigg THEN
      nPIDExeSkipCounter:=nPIDExeSkipCounter + 1;
	  
      IF nPIDExeSkipCounter >= GVL_Parameters.nPhasePIDReducedSampleRateFactor THEN
		//Limit output velocity difference from nominal
        IF(fPhaseErrorFiltered > 0) THEN  //Pos error
          IF ABS(fPhaseErrorFiltered)>15 THEN
            fDeltaVelo:= 0.005;
          ELSIF ABS(fPhaseErrorFiltered)>4 THEN
            fDeltaVelo:= 0.003;
          ELSIF ABS(fPhaseErrorFiltered)>1 THEN
            fDeltaVelo:= 0.0017;
          ELSIF ABS(fPhaseErrorFiltered)>0.5 THEN
            fDeltaVelo:= 0.0012;
          ELSE
	        fDeltaVelo:= 0.001;
          END_IF
        ELSE // neg error
          IF ABS(fPhaseErrorFiltered)>15 THEN  
            fDeltaVelo:= 0.005;
          ELSIF ABS(fPhaseErrorFiltered)>4 THEN
            fDeltaVelo:= 0.003;
          ELSIF ABS(fPhaseErrorFiltered)>1 THEN
            fDeltaVelo:= 0.003;
          ELSIF ABS(fPhaseErrorFiltered)>0.5 THEN
            fDeltaVelo:= 0.003;
          ELSE
	        fDeltaVelo:= 0.0025;
          END_IF	
        END_IF
        nPIDExeSkipCounter:=0;
        fbPhasePID(fSetpointValue:=0,
                   fActualValue := fPhaseErrorFiltered,
                   bReset       := bPhaseControlReset,
		  	       fFF          := 0,
			       fKp          := fPhaseControlKp,
			       fKi          := fPhaseControlKi,
			       fKd          := fPhaseControlKd,
			       fKff         := fPhaseControlKff,
			       fIOutputMin  :=-fDeltaVelo*0.65,
			       fIOutputMax  := fDeltaVelo*0.65,
			       fOutputMin   := -fDeltaVelo,
			       fOutputMax   := fDeltaVelo);
        fPidAdd:=fbPhasePID.fCtrlOutput;
      END_IF
    ELSIF NOT bPhaseAlgTrigg THEN
      fbPhasePID(bReset:=TRUE);  //Reset pid since not used
      fPidAdd:=0;
    END_IF
	fSpeedSetpointLocal:=fNomSpeedSetAdjust+fPidAdd;
	
  E_PHASE_TYPE.SUPERIMPOSE:  
    // Phasing using position superimpose block
	// Positioning is overeloaded over the constant velocity command
	
    //Limit output velocity difference from nominal
    IF(fPhaseErrorFiltered > 0) THEN  //Pos error
      IF ABS(fPhaseErrorFiltered)>15 THEN
        fDeltaVelo:= 0.005;
      ELSIF ABS(fPhaseErrorFiltered)>4 THEN
        fDeltaVelo:= 0.003;
      ELSIF ABS(fPhaseErrorFiltered)>1 THEN
        fDeltaVelo:= 0.002;
      ELSIF ABS(fPhaseErrorFiltered)>0.5 THEN
        fDeltaVelo:= 0.0015;
      ELSE
        fDeltaVelo:= 0.0015;
      END_IF
    ELSE // neg error
      IF ABS(fPhaseErrorFiltered)>15 THEN  
        fDeltaVelo:= 0.005;
      ELSIF ABS(fPhaseErrorFiltered)>4 THEN
        fDeltaVelo:= 0.0035;
      ELSIF ABS(fPhaseErrorFiltered)>1 THEN
        fDeltaVelo:= 0.0035;
      ELSIF ABS(fPhaseErrorFiltered)>0.5 THEN
        fDeltaVelo:= 0.0035;
      ELSE
	    fDeltaVelo:= 0.0025;
      END_IF	
    END_IF  
	fbSuperImpose(bExecute:=bExecuteSuperImpose AND bPhaseAlgTrigg,
                  iSampleRateMs:=GVL_Parameters.nTaskSampleTime,
                  fNominalVelocityRpm:=fNomSpeedSetAdjust,
                  fMaxDeltaVelocityRpm:=fDeltaVelo,
                  fPhaseErrorDeg:=fPhaseErrorFiltered/(GVL_Parameters.fWheelDiameter*pi)*360);
 
    fSpeedSetpointLocal:=fbSuperImpose.fVelocitySetpointRpm;
	fbPhasePID(bReset:=TRUE);  //Reset pid since not used
	
  E_PHASE_TYPE.ONLY_MEASURE:  
    // No control, just measure phase error.
	// Usefull for tuning nominal speed.
	// Procedure: 
	// 1: Set to "ONLY_MEASURE" mode
	// 2: ramp up to nominal speed
	// 3: at constant speed adjust GVL_Parameters.fNominalSpeedAdjust so that
	//    phase error is not changing.
	//    -if phase error is increasing then increase velocity
	//    -if phase error is decreasing then decrease velocity 
 
    fSpeedSetpointLocal:=fNomSpeedSetAdjust;
	fbPhasePID(bReset:=TRUE);  //Reset pid since not used
  ELSE
	fSpeedSetpointLocal:=0;
	fbPhasePID(bReset:=TRUE);  //Reset pid since not used
END_CASE;

fbPWM(
       En:=TRUE,
       bEnable:=TRUE,
       iBlockSampleTimeMicroS:=GVL_Parameters.nTaskSampleTime*1000,
       iProcessSampleTimeMicroS:=71000*GVL_Parameters.nPhasePIDReducedSampleRateFactor,
       iDecimalPoint:=3,
       fInput:=fSpeedSetpointLocal,
       bPromoteHigh:=fPhaseErrorFiltered>0,
       ePwmType:=ePwmType);

fSpeedSetpoint:=fbPWM.fOutput;

IF fSpeedSetpoint>GVL_Parameters.fMaximumSPeedRpm THEN
  fSpeedSetpoint:=GVL_Parameters.fMaximumSPeedRpm; 
END_IF

IF NOT bExecute THEN
  fSpeedSetpoint:=0;	
END_IF

dLatchedPositionOld:=dLatchedPosition;
 
//*********Errorhandling
// Latched pulses missing
IF nMissedTimingPulsesOld<>nMissedTimingPulses THEN
  bError:=TRUE;
  nErrorId:=GVL_ErrorCodes.nErrorNoLatchId;
  sErrorStr:=GVL_ErrorCodes.sErrorNoLatchStr;
END_IF

(*IF nMissedTimingPulsesLowOld<>nMissedTimingPulsesLow THEN
  bError:=TRUE;
  nErrorId:=GVL_ErrorCodes.nErrorNoLatchId;
  sErrorStr:=GVL_ErrorCodes.sErrorNoLatchStr;
END_IF*)

IF bReset THEN
  bError:=FALSE;
  nErrorId:=0;
  //nMissedTimingPulses:=0;
  timerCheckLatchFreqHigh(IN:=FALSE);  //Reset
END_IF

nMissedTimingPulsesOld:=nMissedTimingPulses;
nMissedTimingPulsesLowold:=nMissedTimingPulsesLow;

END_FUNCTION_BLOCK

